// TIA Portal project "Vaja1" (V13)

(* hardware
DEVICE "S7300/ET200M station_1"  S7-300 station
   slot 0: "Rail_0"  Rail  6ES7 390-1***0-0AA0
   slot 1: "PS 307 2A_1"  PS 307 2A  6ES7 307-1BA00-0AA0
   slot 2: "PLC-236"  CPU 315-2 PN/DP  6ES7 315-2EH13-0AB0  V2.6
      slot 1: "MPI/DP interface_1"  X1
      slot 2: "PROFINET interface_1"  PN-IO
         slot 1: "Port_1"  Port
   slot 4: "DI 16/DO 16x24VDC/0.5A_1"  DI16/DO16 x 24V / 0.5A  6ES7 323-1BL00-0AA0
DEVICE "PC station"  SIMATIC PC station
   slot 0: "PC station"  Rail  SIMATIC PC-Station  V1.0
      slot 125: "Stationmanager"  Station_Manager  V6.0.4
   slot 1: "IE general_1"  IE General  IE_CP  V8.2.0
   slot 3: "HMI_RT_1"  WinCC RT Advanced  6AV2 104-0xxxx-xxxx  13.0.1.0
      slot 33792: "Host interface"  Host interface
*)

// ===== PLC "PLC-236"  CPU 315-2 PN/DP =====

VAR_GLOBAL   // PLC tag table "Default tag table"
   "rdeca_levo_potiskac_B_smer_0_nazaj_1_naprej" AT %Q1.4 : Bool;
   "rumena_levo_potiskac_B_premikanje" AT %Q1.5 : Bool;
   "rdeca_desno_tekoci_trak_B_izhod_smer_0_nazaj_1_naprej" AT %Q1.6 : Bool;
   "rumena_desno_tekoci_trak_B_izhod_premikanje" AT %Q1.7 : Bool;
   "kljuc" AT %I1.2 : Bool;
   "zelena" AT %I1.3 : Bool;
   "crna_levo_zgoraj" AT %I1.4 : Bool;
   "crna_levo_spodaj" AT %I1.5 : Bool;
   "crna_desno_zgoraj" AT %I1.6 : Bool;
   "crna_desno_spodaj" AT %I1.7 : Bool;
   "fotocelica_material_na_vhodu_NC" AT %I0.0 : Bool;
   "fotocelica_materal_pred_potiskacem_NC" AT %I0.1 : Bool;
   "potiskac_A_koncni_polozaj_spredaj_NO" AT %I0.2 : Bool;
   "potiskac_A_koncni_polozaj_zadaj_NO" AT %I0.3 : Bool;
   "fotocelica_material_pod_napravo_A_NC" AT %I0.4 : Bool;
   "fotocelica_material_pod_napravo_B_NC" AT %I0.5 : Bool;
   "potiskac_B_koncni_polozaj_zadaj_NO" AT %I0.6 : Bool;
   "potiskac_B_koncni_polozaj_spredaj_NO" AT %I0.7 : Bool;
   "fotocelica_material_na_izhodu_NC" AT %I1.0 : Bool;
   "potiskac_A_smer_0_nazaj_1_naprej" AT %Q0.0 : Bool;
   "potiskac_A_premikanje" AT %Q0.1 : Bool;
   "trak_A_vhod_smer_0_naprej_1_nazaj" AT %Q0.2 : Bool;
   "trak_A_vhod_premikanje" AT %Q0.3 : Bool;
   "trak_A_stroj_smer_0_nazaj_1_naprej" AT %Q0.4 : Bool;
   "trak_A_stroj_premikanje" AT %Q0.5 : Bool;
   "naprava_A_smer_0_CW_1_CCW" AT %Q0.6 : Bool;
   "naprava_A_premikanje" AT %Q0.7 : Bool;
   "naprava_B_smer_0_CW_1_CCW" AT %Q1.0 : Bool;
   "naprava_B_premikanje" AT %Q1.1 : Bool;
   "trak_B_stroj_smer_0_naprej_1_nazaj" AT %Q1.2 : Bool;
   "trak_B_stroj_premikanje" AT %Q1.3 : Bool;
   "retval" AT %MW2 : Int;
   "Startup_Flag" AT %M0.1 : Bool;
   "Ready_Flag" AT %M0.2 : Bool;
   "Clock_10Hz" AT %M5.0 : Bool;
   "Pause_Motors_Flag" AT %M0.3 : Bool;
END_VAR

TYPE "Lokacija"
   STRUCT
      ID : Int;
      zasedenost : Bool;
      senzor : Bool;
      recept : "Recept";
      premikanje : Bool;
   END_STRUCT;
END_TYPE

TYPE "Recept"
   STRUCT
      vrtanje1 : Bool;
      ID_recepta : Int;
      cas_vrtanja1 : Time;
      vrtanje2 : Bool;
      cas_vrtanja2 : Time;
      smer_1 : Bool;
      smer_2 : Bool;
   END_STRUCT;
END_TYPE

// folder: AktivacijaIzvrsnihClenov

DATA_BLOCK "Izhodi"   // DB5
{ S7_Optimized_Access := 'FALSE' }
VERSION : 0.1
   VAR
      potiskac_A_smer : Bool;
      potiskac_A_premikanje : Bool;
      trak_A_vhod_smer : Bool;
      trak_A_vhod_premikanje : Bool;
      trak_A_stroj_smer : Bool;
      trak_A_stroj_premikanje : Bool;
      naprava_A_smer : Bool;
      naprava_A_premikanje : Bool;
      naprava_B_smer : Bool;
      naprava_B_premikanje : Bool;
      trak_B_stroj_smer : Bool;
      trak_B_stroj_premikanje : Bool;
      rdeca_levo_potiskac_B_smer : Bool;
      rumena_levo_potiskac_B_premikanje : Bool;
      rdeca_desno_tekoci_trak_B_izhod_smer : Bool;
      rumena_desno_tekoci_trak_B_izhod_premikanje : Bool;
   END_VAR
BEGIN
END_DATA_BLOCK

// folder: BranjeSenzorjev

DATA_BLOCK "Senzorji_DB"   // DB4
{ S7_Optimized_Access := 'FALSE' }
VERSION : 0.1
   VAR
      fotocelica_material_na_vhodu : Bool;
      fotocelica_materal_pred_potiskacem : Bool;
      navidezni_potiskac_A : Bool;
      potiskac_A_koncni_polozaj_spredaj : Bool;
      potiskac_A_koncni_polozaj_zadaj : Bool;
      fotocelica_material_pod_napravo_A : Bool;
      fotocelica_material_pod_napravo_B : Bool;
      navidezni_potiskac_B : Bool;
      potiskac_B_koncni_polozaj_zadaj : Bool;
      potiskac_B_koncni_polozaj_spredaj : Bool;
      fotocelica_material_na_izhodu : Bool;
      kljuc : Bool;
      zelena_tipka : Bool;
      crna_levo_zgoraj : Bool;
      crna_levo_spodaj : Bool;
      crna_desno_zgoraj : Bool;
      crna_desno_spodaj : Bool;
   END_VAR
BEGIN
END_DATA_BLOCK

// folder: GlavniProgram

DATA_BLOCK "AutoMotorji"   // DB6
{ S7_Optimized_Access := 'FALSE' }
VERSION : 0.1
   VAR
      potiskac_A_naprej : Bool;
      potiskac_A_nazaj : Bool;
      trak_A_vhod_naprej : Bool;
      trak_A_vhod_nazaj : Bool;
      trak_A_stroj_naprej : Bool;
      trak_A_stroj_nazaj : Bool;
      naprava_A_CW : Bool;
      naprava_A_CCW : Bool;
      naprava_B_CW : Bool;
      naprava_B_CCW : Bool;
      trak_B_stroj_naprej : Bool;
      trak_B_stroj_nazaj : Bool;
      potiskac_B_naprej : Bool;
      potiskac_B_nazaj : Bool;
      trak_B_izhod_naprej : Bool;
      trak_B_izhod_nazaj : Bool;
   END_VAR
BEGIN
END_DATA_BLOCK

DATA_BLOCK "Auto_0_vhod1_DB"   // DB8
{ S7_Optimized_Access := 'FALSE' }
VERSION : 0.1
// stored: InstanceOfName Auto_0_vhod1
"Auto_0_vhod1"
BEGIN
END_DATA_BLOCK

DATA_BLOCK "Auto_1_Potiskac_DB"   // DB10
{ S7_Optimized_Access := 'FALSE' }
VERSION : 0.1
// stored: InstanceOfName Auto_1_Potiskac
"Auto_1_Potiskac"
BEGIN
END_DATA_BLOCK

DATA_BLOCK "Auto_2_A_Naprava_DB"   // DB11
{ S7_Optimized_Access := 'FALSE' }
VERSION : 0.1
// stored: InstanceOfName Auto_2_A_Naprava
"Auto_2_A_Naprava"
BEGIN
END_DATA_BLOCK

DATA_BLOCK "Auto_3_B_Naprava_DB"   // DB13
{ S7_Optimized_Access := 'FALSE' }
VERSION : 0.1
// stored: InstanceOfName Auto_3_B_Naprava
"Auto_3_B_Naprava"
BEGIN
END_DATA_BLOCK

DATA_BLOCK "Auto_4_Potiskac_DB"   // DB14
{ S7_Optimized_Access := 'FALSE' }
VERSION : 0.1
// stored: InstanceOfName Auto_4_Potiskac
"Auto_4_Potiskac"
BEGIN
END_DATA_BLOCK

DATA_BLOCK "Auto_5_Izhod_DB"   // DB15
{ S7_Optimized_Access := 'FALSE' }
VERSION : 0.1
// stored: InstanceOfName Auto_5_Izhod
"Auto_5_Izhod"
BEGIN
END_DATA_BLOCK

// folder: GlavniProgram/Alarmi

DATA_BLOCK "Alarmi_DB"   // DB18
{ S7_Optimized_Access := 'FALSE' }
VERSION : 0.1
// stored: InstanceOfName Alarmi
"Alarmi"
BEGIN
END_DATA_BLOCK

// folder: GlavniProgram/SCADA

DATA_BLOCK "SCADA"   // DB16
{ S7_Optimized_Access := 'FALSE' }
VERSION : 0.1
   VAR
      alarmi : Array[0..15] of Bool;
      alarm_aktiven_globalno : Bool;
      recept_num : Int;
      alarm_potrditev : Bool;
      recept : "Recept";
   END_VAR
BEGIN
END_DATA_BLOCK

DATA_BLOCK "SCADAVisual_DB"   // DB23
{ S7_Optimized_Access := 'FALSE' }
VERSION : 0.1
// stored: InstanceOfName SCADAVisual
"SCADAVisual"
BEGIN
END_DATA_BLOCK

// folder: MotorLogic

DATA_BLOCK "Izbira_motorja_DB"   // DB1
{ S7_Optimized_Access := 'FALSE' }
VERSION : 0.1
// stored: InstanceOfName Izbira_motorja
"Izbira_motorja"
BEGIN
END_DATA_BLOCK

DATA_BLOCK "Motorji_DB"   // DB2
{ S7_Optimized_Access := 'FALSE' }
VERSION : 0.1
// stored: InstanceOfName Motorji
"Motorji"
BEGIN
END_DATA_BLOCK

// folder: SledenjeMateriala

DATA_BLOCK "Lokacije_DB"   // DB3
{ S7_Optimized_Access := 'FALSE' }
VERSION : 0.1
   VAR
      L1_vhod_1 : "Lokacija";
      L2_vhod_2 : "Lokacija";
      L3_potiskac_A : "Lokacija";
      L4_naprava_A : "Lokacija";
      L5_naprava_B : "Lokacija";
      L6_potiskac_B : "Lokacija";
      L7_izhod : "Lokacija";
      Empty : "Lokacija";
   END_VAR
BEGIN
END_DATA_BLOCK

// folder: (top level)

ORGANIZATION_BLOCK "Main"   // OB1, LAD
TITLE = "Main Program Sweep (Cycle)"
{ S7_Optimized_Access := 'FALSE' }
VERSION : 0.1
BEGIN

REGION Network 1: Rocno vodenje
   // nc ne bo komentar
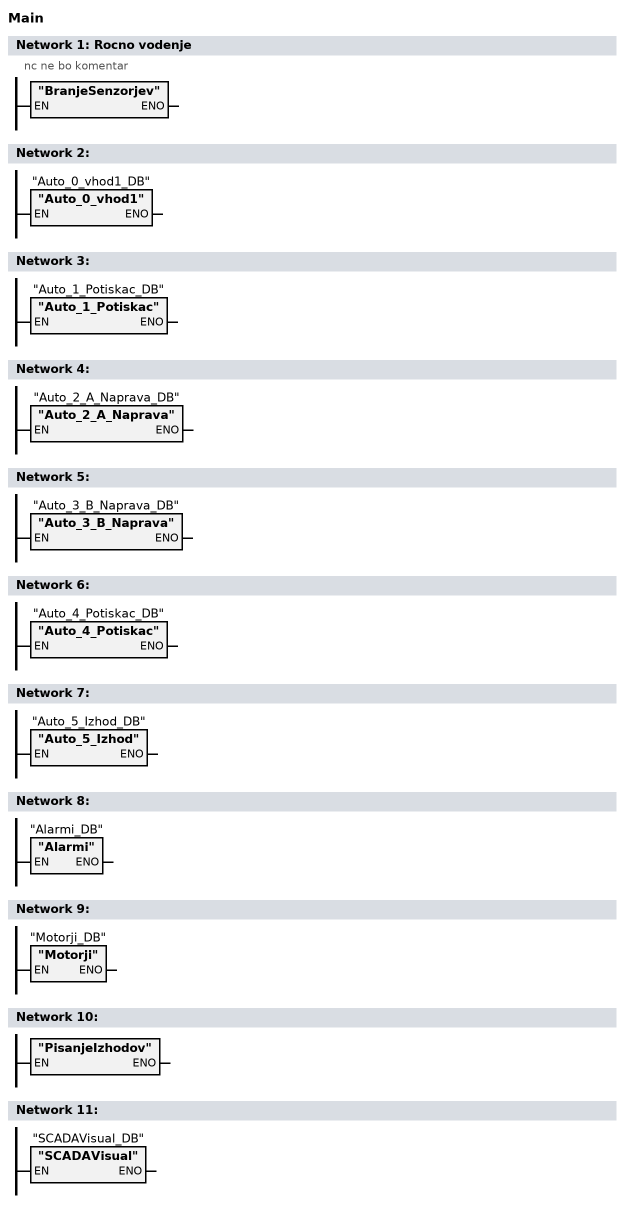
   RUNG wire#powerrail
      "BranjeSenzorjev"()
   END_RUNG
   // the same network as SCL:
   "BranjeSenzorjev"();
END_REGION

REGION Network 2
   RUNG wire#powerrail
      "Auto_0_vhod1_DB"()
   END_RUNG
   // the same network as SCL:
   "Auto_0_vhod1_DB"();   // "Auto_0_vhod1"
END_REGION

REGION Network 3
   RUNG wire#powerrail
      "Auto_1_Potiskac_DB"()
   END_RUNG
   // the same network as SCL:
   "Auto_1_Potiskac_DB"();   // "Auto_1_Potiskac"
END_REGION

REGION Network 4
   RUNG wire#powerrail
      "Auto_2_A_Naprava_DB"()
   END_RUNG
   // the same network as SCL:
   "Auto_2_A_Naprava_DB"();   // "Auto_2_A_Naprava"
END_REGION

REGION Network 5
   RUNG wire#powerrail
      "Auto_3_B_Naprava_DB"()
   END_RUNG
   // the same network as SCL:
   "Auto_3_B_Naprava_DB"();   // "Auto_3_B_Naprava"
END_REGION

REGION Network 6
   RUNG wire#powerrail
      "Auto_4_Potiskac_DB"()
   END_RUNG
   // the same network as SCL:
   "Auto_4_Potiskac_DB"();   // "Auto_4_Potiskac"
END_REGION

REGION Network 7
   RUNG wire#powerrail
      "Auto_5_Izhod_DB"()
   END_RUNG
   // the same network as SCL:
   "Auto_5_Izhod_DB"();   // "Auto_5_Izhod"
END_REGION

REGION Network 8
   RUNG wire#powerrail
      "Alarmi_DB"()
   END_RUNG
   // the same network as SCL:
   "Alarmi_DB"();   // "Alarmi"
END_REGION

REGION Network 9
   RUNG wire#powerrail
      "Motorji_DB"()
   END_RUNG
   // the same network as SCL:
   "Motorji_DB"();   // "Motorji"
END_REGION

REGION Network 10
   RUNG wire#powerrail
      "PisanjeIzhodov"()
   END_RUNG
   // the same network as SCL:
   "PisanjeIzhodov"();
END_REGION

REGION Network 11
   RUNG wire#powerrail
      "SCADAVisual_DB"()
   END_RUNG
   // the same network as SCL:
   "SCADAVisual_DB"();   // "SCADAVisual"
END_REGION
END_ORGANIZATION_BLOCK

// folder: AktivacijaIzvrsnihClenov

FUNCTION "PisanjeIzhodov" : Void   // FC2, LAD
TITLE = Pisanje iz podatkovne baze na izhode.
{ S7_Optimized_Access := 'FALSE' }
VERSION : 0.1
BEGIN

REGION Network 1: Potiskač A smer.
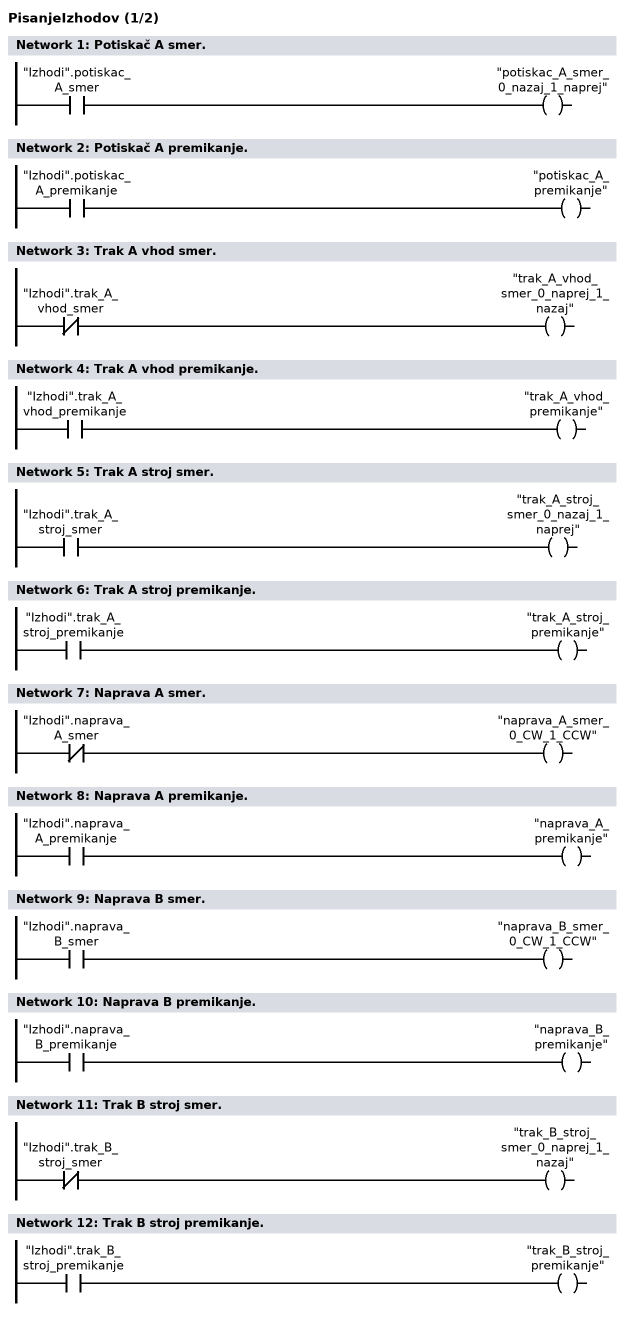
   RUNG wire#powerrail
      Contact( "Izhodi".potiskac_A_smer )
      Coil( "potiskac_A_smer_0_nazaj_1_naprej" )
   END_RUNG
   // the same network as SCL:
   "potiskac_A_smer_0_nazaj_1_naprej" := "Izhodi".potiskac_A_smer;
END_REGION

REGION Network 2: Potiskač A premikanje.
   RUNG wire#powerrail
      Contact( "Izhodi".potiskac_A_premikanje )
      Coil( "potiskac_A_premikanje" )
   END_RUNG
   // the same network as SCL:
   "potiskac_A_premikanje" := "Izhodi".potiskac_A_premikanje;
END_REGION

REGION Network 3: Trak A vhod smer.
   RUNG wire#powerrail
      I_Contact( "Izhodi".trak_A_vhod_smer )
      Coil( "trak_A_vhod_smer_0_naprej_1_nazaj" )
   END_RUNG
   // the same network as SCL:
   "trak_A_vhod_smer_0_naprej_1_nazaj" := NOT "Izhodi".trak_A_vhod_smer;
END_REGION

REGION Network 4: Trak A vhod premikanje.
   RUNG wire#powerrail
      Contact( "Izhodi".trak_A_vhod_premikanje )
      Coil( "trak_A_vhod_premikanje" )
   END_RUNG
   // the same network as SCL:
   "trak_A_vhod_premikanje" := "Izhodi".trak_A_vhod_premikanje;
END_REGION

REGION Network 5: Trak A stroj smer.
   RUNG wire#powerrail
      Contact( "Izhodi".trak_A_stroj_smer )
      Coil( "trak_A_stroj_smer_0_nazaj_1_naprej" )
   END_RUNG
   // the same network as SCL:
   "trak_A_stroj_smer_0_nazaj_1_naprej" := "Izhodi".trak_A_stroj_smer;
END_REGION

REGION Network 6: Trak A stroj premikanje.
   RUNG wire#powerrail
      Contact( "Izhodi".trak_A_stroj_premikanje )
      Coil( "trak_A_stroj_premikanje" )
   END_RUNG
   // the same network as SCL:
   "trak_A_stroj_premikanje" := "Izhodi".trak_A_stroj_premikanje;
END_REGION

REGION Network 7: Naprava A smer.
   RUNG wire#powerrail
      I_Contact( "Izhodi".naprava_A_smer )
      Coil( "naprava_A_smer_0_CW_1_CCW" )
   END_RUNG
   // the same network as SCL:
   "naprava_A_smer_0_CW_1_CCW" := NOT "Izhodi".naprava_A_smer;
END_REGION

REGION Network 8: Naprava A premikanje.
   RUNG wire#powerrail
      Contact( "Izhodi".naprava_A_premikanje )
      Coil( "naprava_A_premikanje" )
   END_RUNG
   // the same network as SCL:
   "naprava_A_premikanje" := "Izhodi".naprava_A_premikanje;
END_REGION

REGION Network 9: Naprava B smer.
   RUNG wire#powerrail
      Contact( "Izhodi".naprava_B_smer )
      Coil( "naprava_B_smer_0_CW_1_CCW" )
   END_RUNG
   // the same network as SCL:
   "naprava_B_smer_0_CW_1_CCW" := "Izhodi".naprava_B_smer;
END_REGION

REGION Network 10: Naprava B premikanje.
   RUNG wire#powerrail
      Contact( "Izhodi".naprava_B_premikanje )
      Coil( "naprava_B_premikanje" )
   END_RUNG
   // the same network as SCL:
   "naprava_B_premikanje" := "Izhodi".naprava_B_premikanje;
END_REGION

REGION Network 11: Trak B stroj smer.
   RUNG wire#powerrail
      I_Contact( "Izhodi".trak_B_stroj_smer )
      Coil( "trak_B_stroj_smer_0_naprej_1_nazaj" )
   END_RUNG
   // the same network as SCL:
   "trak_B_stroj_smer_0_naprej_1_nazaj" := NOT "Izhodi".trak_B_stroj_smer;
END_REGION

REGION Network 12: Trak B stroj premikanje.
   RUNG wire#powerrail
      Contact( "Izhodi".trak_B_stroj_premikanje )
      Coil( "trak_B_stroj_premikanje" )
   END_RUNG
   // the same network as SCL:
   "trak_B_stroj_premikanje" := "Izhodi".trak_B_stroj_premikanje;
END_REGION

REGION Network 13: Potiskač B smer.
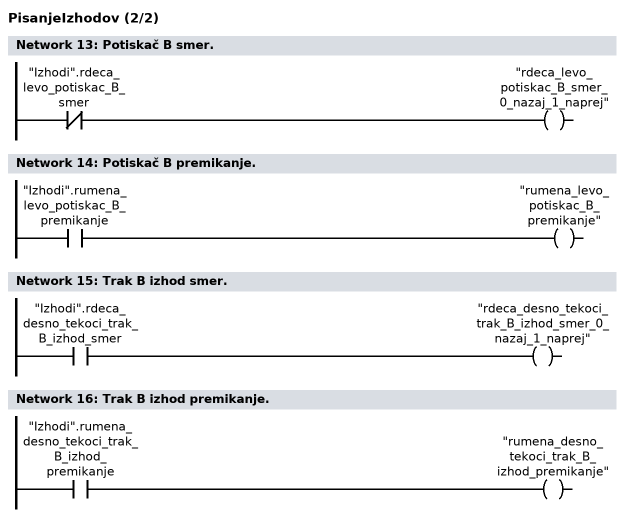
   RUNG wire#powerrail
      I_Contact( "Izhodi".rdeca_levo_potiskac_B_smer )
      Coil( "rdeca_levo_potiskac_B_smer_0_nazaj_1_naprej" )
   END_RUNG
   // the same network as SCL:
   "rdeca_levo_potiskac_B_smer_0_nazaj_1_naprej" := NOT "Izhodi".rdeca_levo_potiskac_B_smer;
END_REGION

REGION Network 14: Potiskač B premikanje.
   RUNG wire#powerrail
      Contact( "Izhodi".rumena_levo_potiskac_B_premikanje )
      Coil( "rumena_levo_potiskac_B_premikanje" )
   END_RUNG
   // the same network as SCL:
   "rumena_levo_potiskac_B_premikanje" := "Izhodi".rumena_levo_potiskac_B_premikanje;
END_REGION

REGION Network 15: Trak B izhod smer.
   RUNG wire#powerrail
      Contact( "Izhodi".rdeca_desno_tekoci_trak_B_izhod_smer )
      Coil( "rdeca_desno_tekoci_trak_B_izhod_smer_0_nazaj_1_naprej" )
   END_RUNG
   // the same network as SCL:
   "rdeca_desno_tekoci_trak_B_izhod_smer_0_nazaj_1_naprej" := "Izhodi".rdeca_desno_tekoci_trak_B_izhod_smer;
END_REGION

REGION Network 16: Trak B izhod premikanje.
   RUNG wire#powerrail
      Contact( "Izhodi".rumena_desno_tekoci_trak_B_izhod_premikanje )
      Coil( "rumena_desno_tekoci_trak_B_izhod_premikanje" )
   END_RUNG
   // the same network as SCL:
   "rumena_desno_tekoci_trak_B_izhod_premikanje" := "Izhodi".rumena_desno_tekoci_trak_B_izhod_premikanje;
END_REGION
END_FUNCTION

// folder: BranjeSenzorjev

FUNCTION "BranjeSenzorjev" : Void   // FC1, LAD
TITLE = Prepis iz vhodov v podatkovno bazo.
{ S7_Optimized_Access := 'FALSE' }
VERSION : 0.1
// Normaliziranje vseh senzorjev (NC/NO).
BEGIN

REGION Network 1: Fotocelica: material na vhodu.
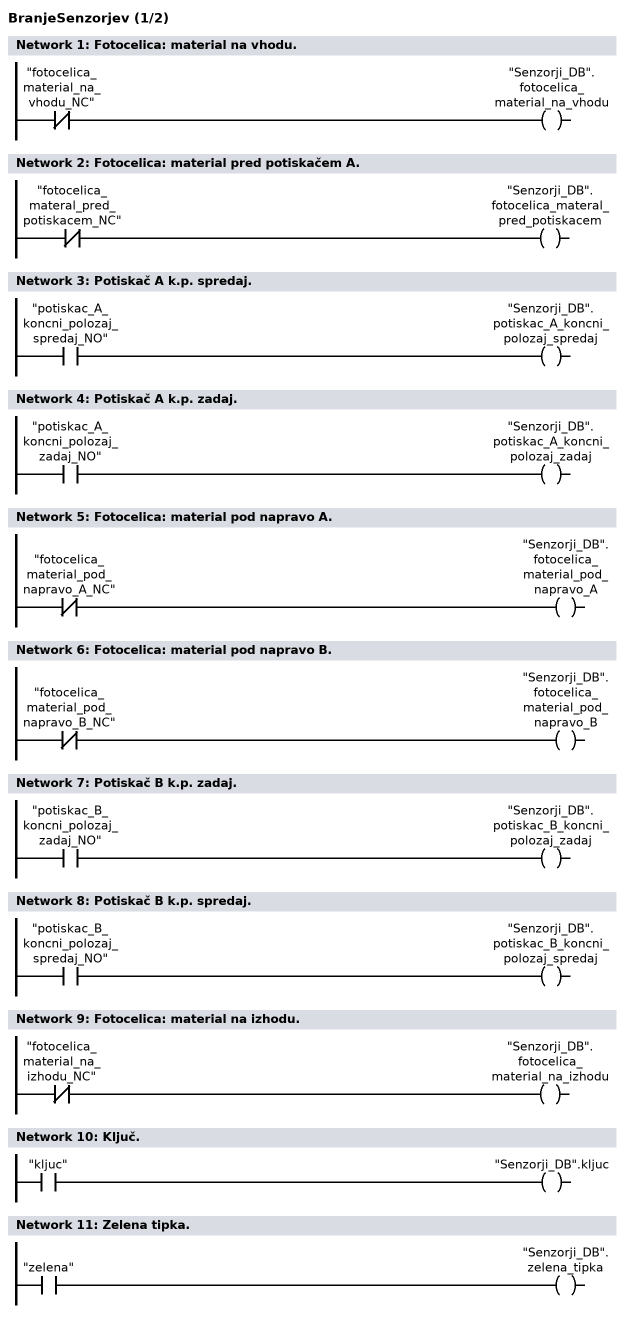
   RUNG wire#powerrail
      I_Contact( "fotocelica_material_na_vhodu_NC" )
      Coil( "Senzorji_DB".fotocelica_material_na_vhodu )
   END_RUNG
   // the same network as SCL:
   "Senzorji_DB".fotocelica_material_na_vhodu := NOT "fotocelica_material_na_vhodu_NC";
END_REGION

REGION Network 2: Fotocelica: material pred potiskačem A.
   RUNG wire#powerrail
      I_Contact( "fotocelica_materal_pred_potiskacem_NC" )
      Coil( "Senzorji_DB".fotocelica_materal_pred_potiskacem )
   END_RUNG
   // the same network as SCL:
   "Senzorji_DB".fotocelica_materal_pred_potiskacem := NOT "fotocelica_materal_pred_potiskacem_NC";
END_REGION

REGION Network 3: Potiskač A k.p. spredaj.
   RUNG wire#powerrail
      Contact( "potiskac_A_koncni_polozaj_spredaj_NO" )
      Coil( "Senzorji_DB".potiskac_A_koncni_polozaj_spredaj )
   END_RUNG
   // the same network as SCL:
   "Senzorji_DB".potiskac_A_koncni_polozaj_spredaj := "potiskac_A_koncni_polozaj_spredaj_NO";
END_REGION

REGION Network 4: Potiskač A k.p. zadaj.
   RUNG wire#powerrail
      Contact( "potiskac_A_koncni_polozaj_zadaj_NO" )
      Coil( "Senzorji_DB".potiskac_A_koncni_polozaj_zadaj )
   END_RUNG
   // the same network as SCL:
   "Senzorji_DB".potiskac_A_koncni_polozaj_zadaj := "potiskac_A_koncni_polozaj_zadaj_NO";
END_REGION

REGION Network 5: Fotocelica: material pod napravo A.
   RUNG wire#powerrail
      I_Contact( "fotocelica_material_pod_napravo_A_NC" )
      Coil( "Senzorji_DB".fotocelica_material_pod_napravo_A )
   END_RUNG
   // the same network as SCL:
   "Senzorji_DB".fotocelica_material_pod_napravo_A := NOT "fotocelica_material_pod_napravo_A_NC";
END_REGION

REGION Network 6: Fotocelica: material pod napravo B.
   RUNG wire#powerrail
      I_Contact( "fotocelica_material_pod_napravo_B_NC" )
      Coil( "Senzorji_DB".fotocelica_material_pod_napravo_B )
   END_RUNG
   // the same network as SCL:
   "Senzorji_DB".fotocelica_material_pod_napravo_B := NOT "fotocelica_material_pod_napravo_B_NC";
END_REGION

REGION Network 7: Potiskač B k.p. zadaj.
   RUNG wire#powerrail
      Contact( "potiskac_B_koncni_polozaj_zadaj_NO" )
      Coil( "Senzorji_DB".potiskac_B_koncni_polozaj_zadaj )
   END_RUNG
   // the same network as SCL:
   "Senzorji_DB".potiskac_B_koncni_polozaj_zadaj := "potiskac_B_koncni_polozaj_zadaj_NO";
END_REGION

REGION Network 8: Potiskač B k.p. spredaj.
   RUNG wire#powerrail
      Contact( "potiskac_B_koncni_polozaj_spredaj_NO" )
      Coil( "Senzorji_DB".potiskac_B_koncni_polozaj_spredaj )
   END_RUNG
   // the same network as SCL:
   "Senzorji_DB".potiskac_B_koncni_polozaj_spredaj := "potiskac_B_koncni_polozaj_spredaj_NO";
END_REGION

REGION Network 9: Fotocelica: material na izhodu.
   RUNG wire#powerrail
      I_Contact( "fotocelica_material_na_izhodu_NC" )
      Coil( "Senzorji_DB".fotocelica_material_na_izhodu )
   END_RUNG
   // the same network as SCL:
   "Senzorji_DB".fotocelica_material_na_izhodu := NOT "fotocelica_material_na_izhodu_NC";
END_REGION

REGION Network 10: Ključ.
   RUNG wire#powerrail
      Contact( "kljuc" )
      Coil( "Senzorji_DB".kljuc )
   END_RUNG
   // the same network as SCL:
   "Senzorji_DB".kljuc := "kljuc";
END_REGION

REGION Network 11: Zelena tipka.
   RUNG wire#powerrail
      Contact( "zelena" )
      Coil( "Senzorji_DB".zelena_tipka )
   END_RUNG
   // the same network as SCL:
   "Senzorji_DB".zelena_tipka := "zelena";
END_REGION

REGION Network 12: Črna tipka levo zgoraj.
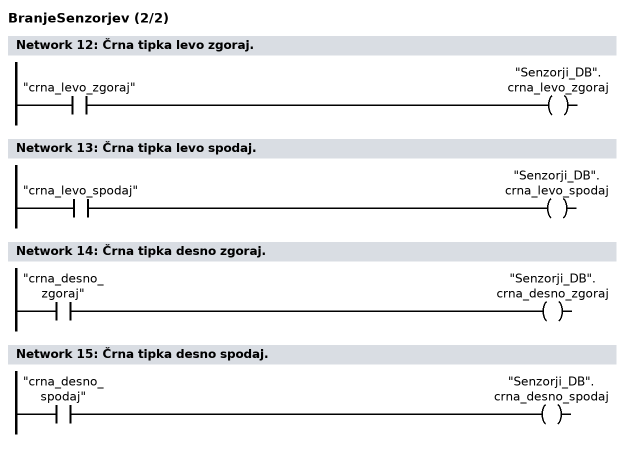
   RUNG wire#powerrail
      Contact( "crna_levo_zgoraj" )
      Coil( "Senzorji_DB".crna_levo_zgoraj )
   END_RUNG
   // the same network as SCL:
   "Senzorji_DB".crna_levo_zgoraj := "crna_levo_zgoraj";
END_REGION

REGION Network 13: Črna tipka levo spodaj.
   RUNG wire#powerrail
      Contact( "crna_levo_spodaj" )
      Coil( "Senzorji_DB".crna_levo_spodaj )
   END_RUNG
   // the same network as SCL:
   "Senzorji_DB".crna_levo_spodaj := "crna_levo_spodaj";
END_REGION

REGION Network 14: Črna tipka desno zgoraj.
   RUNG wire#powerrail
      Contact( "crna_desno_zgoraj" )
      Coil( "Senzorji_DB".crna_desno_zgoraj )
   END_RUNG
   // the same network as SCL:
   "Senzorji_DB".crna_desno_zgoraj := "crna_desno_zgoraj";
END_REGION

REGION Network 15: Črna tipka desno spodaj.
   RUNG wire#powerrail
      Contact( "crna_desno_spodaj" )
      Coil( "Senzorji_DB".crna_desno_spodaj )
   END_RUNG
   // the same network as SCL:
   "Senzorji_DB".crna_desno_spodaj := "crna_desno_spodaj";
END_REGION
END_FUNCTION

// folder: GlavniProgram

FUNCTION_BLOCK "Auto_2_A_Naprava"   // FB4, LAD
TITLE = Stanje 2: Naprava A.
{ S7_Optimized_Access := 'FALSE' }
VERSION : 0.1
// V stanju dve vrtimo napravo A za čas definiran v receptu in smer definirano v receptu, potem material pošljemo do naprave B.
   VAR_TEMP   // added for the SCL form of the ladder/FBD networks
      _w1 : Bool;
      _w2 : Bool;
      _w3 : Bool;
      _w4 : Bool;
      _w5 : Bool;
   END_VAR
BEGIN

REGION Network 1
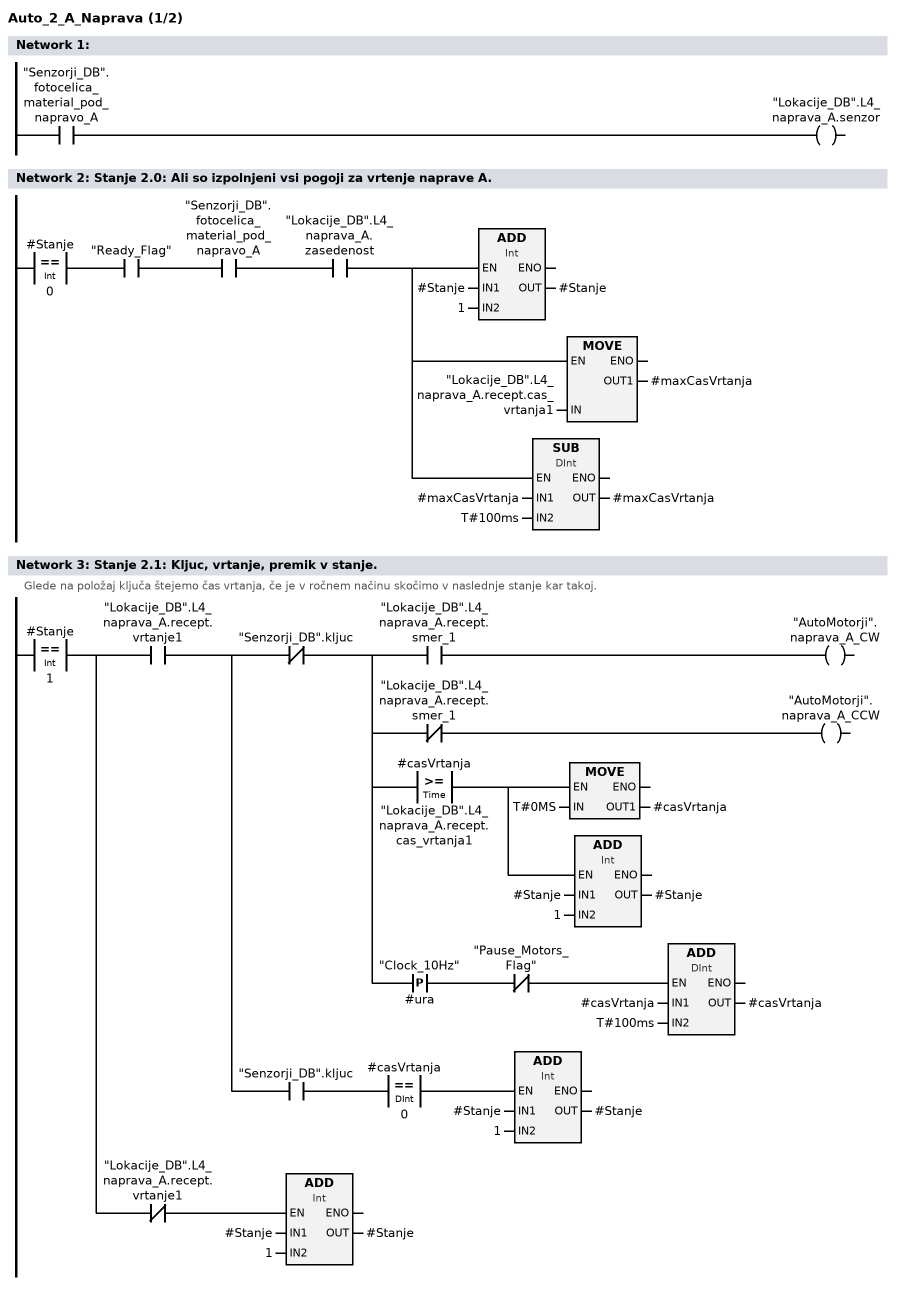
   RUNG wire#powerrail
      Contact( "Senzorji_DB".fotocelica_material_pod_napravo_A )
      Coil( "Lokacije_DB".L4_naprava_A.senzor )
   END_RUNG
   // the same network as SCL:
   "Lokacije_DB".L4_naprava_A.senzor := "Senzorji_DB".fotocelica_material_pod_napravo_A;
END_REGION

REGION Network 2: Stanje 2.0: Ali so izpolnjeni vsi pogoji za vrtenje naprave A.
   RUNG wire#powerrail
      { S7_Templates := "SrcType := Int" } EQ_Contact(in1 := #Stanje, in2 := 0)
      Contact( "Ready_Flag" )
      Contact( "Senzorji_DB".fotocelica_material_pod_napravo_A )
      Contact( "Lokacije_DB".L4_naprava_A.zasedenost )
      wire#w1
      { S7_Templates := "SrcType := Int"; S7_GenerateENO := "TRUE" } Add(in1 := #Stanje, in2 := 1, out => #Stanje)
   END_RUNG
   RUNG wire#w1
      { S7_GenerateENO := "TRUE" } Move(in := "Lokacije_DB".L4_naprava_A.recept.cas_vrtanja1, out1 => #maxCasVrtanja)
   END_RUNG
   RUNG wire#w1
      { S7_Templates := "SrcType := DInt"; S7_GenerateENO := "TRUE" } Sub(in1 := #maxCasVrtanja, in2 := T#100ms, out => #maxCasVrtanja)
   END_RUNG
   // the same network as SCL:
   #_w1 := (#Stanje = 0) AND "Ready_Flag" AND "Senzorji_DB".fotocelica_material_pod_napravo_A AND "Lokacije_DB".L4_naprava_A.zasedenost;
   IF #_w1 THEN
       #Stanje := #Stanje + 1;
       #maxCasVrtanja := "Lokacije_DB".L4_naprava_A.recept.cas_vrtanja1;
       #maxCasVrtanja := #maxCasVrtanja - T#100ms;
   END_IF;
END_REGION

REGION Network 3: Stanje 2.1: Kljuc, vrtanje, premik v stanje.
   // Glede na položaj ključa štejemo čas vrtanja, če je v ročnem načinu skočimo v naslednje stanje kar takoj.
   RUNG wire#powerrail
      { S7_Templates := "SrcType := Int" } EQ_Contact(in1 := #Stanje, in2 := 1)
      wire#w1
      Contact( "Lokacije_DB".L4_naprava_A.recept.vrtanje1 )
      wire#w2
      I_Contact( "Senzorji_DB".kljuc )
      wire#w3
      Contact( "Lokacije_DB".L4_naprava_A.recept.smer_1 )
      Coil( "AutoMotorji".naprava_A_CW )
   END_RUNG
   RUNG wire#w3
      I_Contact( "Lokacije_DB".L4_naprava_A.recept.smer_1 )
      Coil( "AutoMotorji".naprava_A_CCW )
   END_RUNG
   RUNG wire#w3
      { S7_Templates := "SrcType := Time" } GE_Contact(in1 := #casVrtanja, in2 := "Lokacije_DB".L4_naprava_A.recept.cas_vrtanja1)
      wire#w4
      { S7_GenerateENO := "TRUE" } Move(in := T#0MS, out1 => #casVrtanja)
   END_RUNG
   RUNG wire#w4
      { S7_Templates := "SrcType := Int"; S7_GenerateENO := "TRUE" } Add(in1 := #Stanje, in2 := 1, out => #Stanje)
   END_RUNG
   RUNG wire#w3
      P_Contact(operand := "Clock_10Hz", bit := #ura)
      I_Contact( "Pause_Motors_Flag" )
      { S7_Templates := "SrcType := DInt"; S7_GenerateENO := "TRUE" } Add(in1 := #casVrtanja, in2 := T#100ms, out => #casVrtanja)
   END_RUNG
   RUNG wire#w2
      Contact( "Senzorji_DB".kljuc )
      { S7_Templates := "SrcType := DInt" } EQ_Contact(in1 := #casVrtanja, in2 := 0)
      { S7_Templates := "SrcType := Int"; S7_GenerateENO := "TRUE" } Add(in1 := #Stanje, in2 := 1, out => #Stanje)
   END_RUNG
   RUNG wire#w1
      I_Contact( "Lokacije_DB".L4_naprava_A.recept.vrtanje1 )
      { S7_Templates := "SrcType := Int"; S7_GenerateENO := "TRUE" } Add(in1 := #Stanje, in2 := 1, out => #Stanje)
   END_RUNG
   // the same network as SCL:
   #_w1 := #Stanje = 1;
   #_w2 := #_w1 AND "Lokacije_DB".L4_naprava_A.recept.vrtanje1;
   #_w3 := #_w2 AND NOT "Senzorji_DB".kljuc;
   "AutoMotorji".naprava_A_CW := #_w3 AND "Lokacije_DB".L4_naprava_A.recept.smer_1;
   "AutoMotorji".naprava_A_CCW := #_w3 AND NOT "Lokacije_DB".L4_naprava_A.recept.smer_1;
   #_w4 := #_w3 AND (#casVrtanja >= "Lokacije_DB".L4_naprava_A.recept.cas_vrtanja1);
   IF #_w4 THEN
       #casVrtanja := T#0MS;
       #Stanje := #Stanje + 1;
   END_IF;
   #_w5 := #_w3 AND "Clock_10Hz" AND NOT #ura;   // rising edge of "Clock_10Hz"
   #ura := "Clock_10Hz";
   IF #_w5 AND NOT "Pause_Motors_Flag" THEN #casVrtanja := #casVrtanja + T#100ms; END_IF;
   IF #_w2 AND "Senzorji_DB".kljuc AND (#casVrtanja = 0) THEN #Stanje := #Stanje + 1; END_IF;
   IF #_w1 AND NOT "Lokacije_DB".L4_naprava_A.recept.vrtanje1 THEN #Stanje := #Stanje + 1; END_IF;
END_REGION

REGION Network 4: Stanje 2.2: Po koncu vrtanja prižgemo tekoča traka, da pride material pod napravo B.
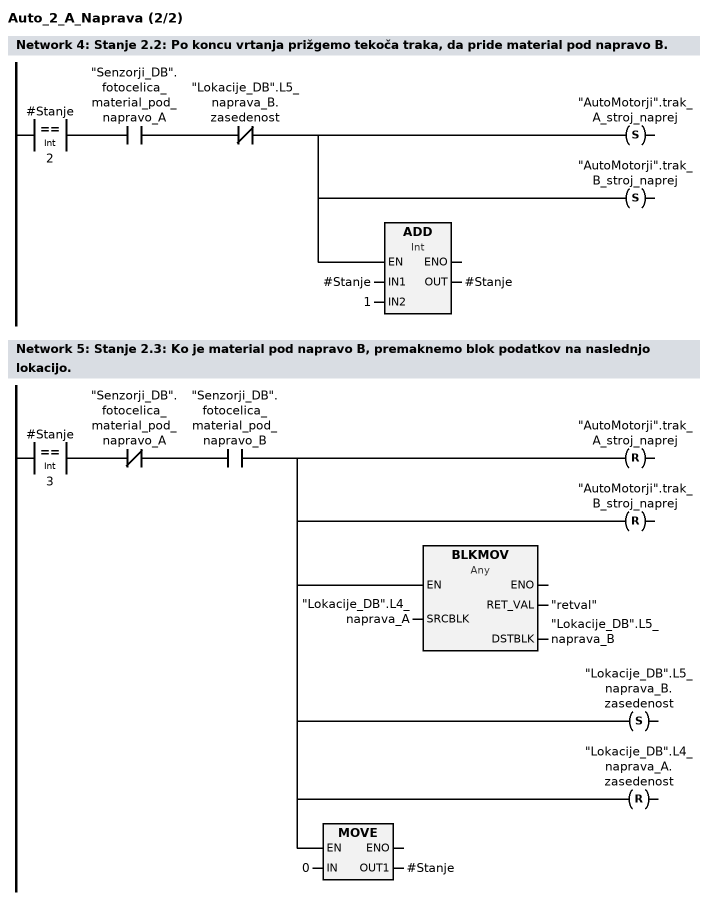
   RUNG wire#powerrail
      { S7_Templates := "SrcType := Int" } EQ_Contact(in1 := #Stanje, in2 := 2)
      Contact( "Senzorji_DB".fotocelica_material_pod_napravo_A )
      I_Contact( "Lokacije_DB".L5_naprava_B.zasedenost )
      wire#w1
      S_Coil( "AutoMotorji".trak_A_stroj_naprej )
   END_RUNG
   RUNG wire#w1
      S_Coil( "AutoMotorji".trak_B_stroj_naprej )
   END_RUNG
   RUNG wire#w1
      { S7_Templates := "SrcType := Int"; S7_GenerateENO := "TRUE" } Add(in1 := #Stanje, in2 := 1, out => #Stanje)
   END_RUNG
   // the same network as SCL:
   IF (#Stanje = 2) AND "Senzorji_DB".fotocelica_material_pod_napravo_A AND NOT "Lokacije_DB".L5_naprava_B.zasedenost THEN
       "AutoMotorji".trak_A_stroj_naprej := TRUE;
       "AutoMotorji".trak_B_stroj_naprej := TRUE;
       #Stanje := #Stanje + 1;
   END_IF;
END_REGION

REGION Network 5: Stanje 2.3: Ko je material pod napravo B, premaknemo blok podatkov na naslednjo lokacijo.
   IF (#Stanje = 3) AND NOT "Senzorji_DB".fotocelica_material_pod_napravo_A AND "Senzorji_DB".fotocelica_material_pod_napravo_B THEN
       "AutoMotorji".trak_A_stroj_naprej := FALSE;
       "AutoMotorji".trak_B_stroj_naprej := FALSE;
   END_IF;
   #_w1 := (#Stanje = 3) AND NOT "Senzorji_DB".fotocelica_material_pod_napravo_A AND "Senzorji_DB".fotocelica_material_pod_napravo_B;
   IF #_w1 THEN
       "retval" := BLKMOV(SRCBLK := "Lokacije_DB".L4_naprava_A, DSTBLK => "Lokacije_DB".L5_naprava_B);
       "Lokacije_DB".L5_naprava_B.zasedenost := TRUE;
       "Lokacije_DB".L4_naprava_A.zasedenost := FALSE;
       #Stanje := 0;
   END_IF;
END_REGION
END_FUNCTION_BLOCK

FUNCTION_BLOCK "Auto_1_Potiskac"   // FB5, LAD
TITLE = Stanje 1 -> potiskač
{ S7_Optimized_Access := 'FALSE' }
VERSION : 0.1
// Premikanje materiala izpred potiskača do drugega tekočega traku.
   VAR_TEMP   // added for the SCL form of the ladder/FBD networks
      _w1 : Bool;
      _w2 : Bool;
      _w3 : Bool;
      _w4 : Bool;
   END_VAR
BEGIN

REGION Network 1: Stanje 1.0: Preverimo ali so vsi pogoji ustrezni za premikanje potiskača.
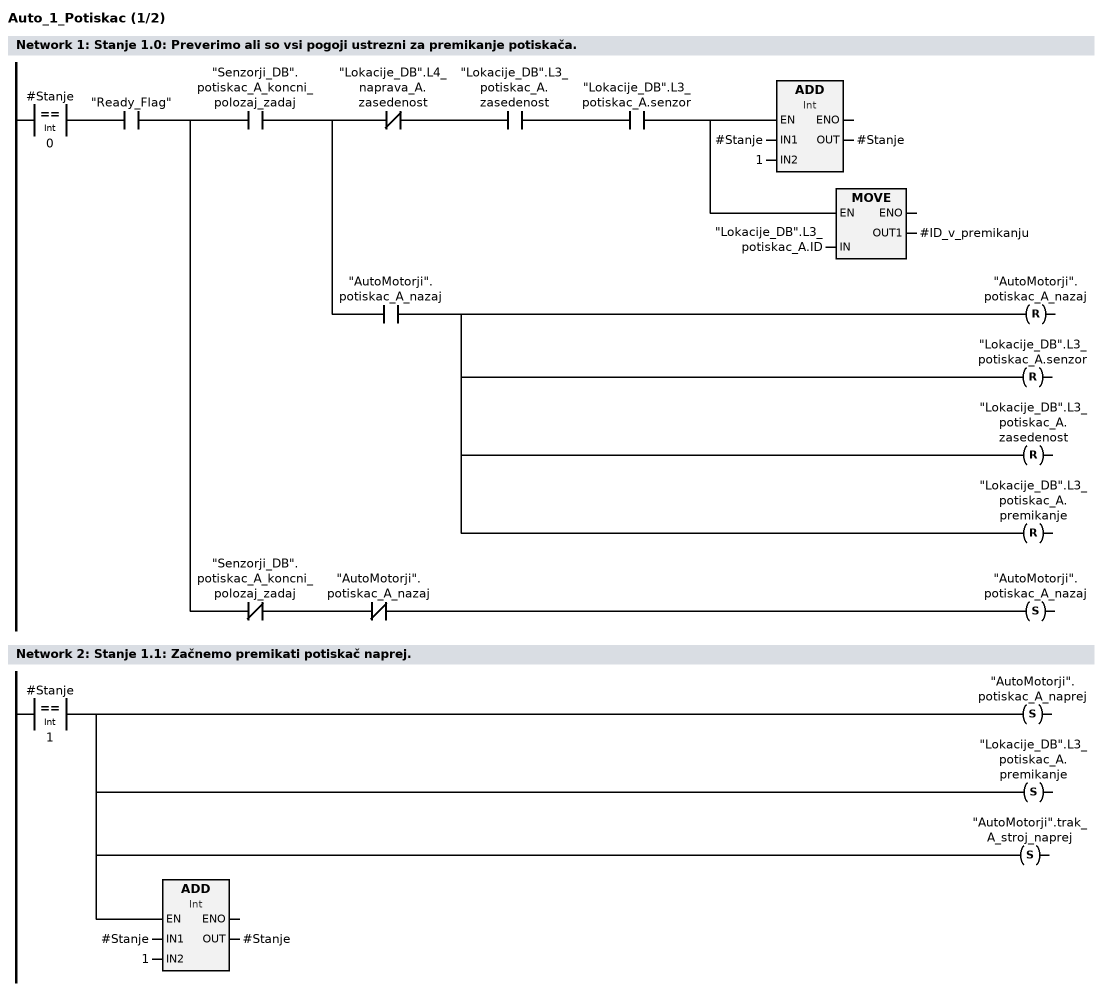
   RUNG wire#powerrail
      { S7_Templates := "SrcType := Int" } EQ_Contact(in1 := #Stanje, in2 := 0)
      Contact( "Ready_Flag" )
      wire#w1
      Contact( "Senzorji_DB".potiskac_A_koncni_polozaj_zadaj )
      wire#w2
      I_Contact( "Lokacije_DB".L4_naprava_A.zasedenost )
      Contact( "Lokacije_DB".L3_potiskac_A.zasedenost )
      Contact( "Lokacije_DB".L3_potiskac_A.senzor )
      wire#w3
      { S7_Templates := "SrcType := Int"; S7_GenerateENO := "TRUE" } Add(in1 := #Stanje, in2 := 1, out => #Stanje)
   END_RUNG
   RUNG wire#w3
      { S7_GenerateENO := "TRUE" } Move(in := "Lokacije_DB".L3_potiskac_A.ID, out1 => #ID_v_premikanju)
   END_RUNG
   RUNG wire#w2
      Contact( "AutoMotorji".potiskac_A_nazaj )
      wire#w4
      R_Coil( "AutoMotorji".potiskac_A_nazaj )
   END_RUNG
   RUNG wire#w4
      R_Coil( "Lokacije_DB".L3_potiskac_A.senzor )
   END_RUNG
   RUNG wire#w4
      R_Coil( "Lokacije_DB".L3_potiskac_A.zasedenost )
   END_RUNG
   RUNG wire#w4
      R_Coil( "Lokacije_DB".L3_potiskac_A.premikanje )
   END_RUNG
   RUNG wire#w1
      I_Contact( "Senzorji_DB".potiskac_A_koncni_polozaj_zadaj )
      I_Contact( "AutoMotorji".potiskac_A_nazaj )
      S_Coil( "AutoMotorji".potiskac_A_nazaj )
   END_RUNG
   // the same network as SCL:
   #_w1 := (#Stanje = 0) AND "Ready_Flag";
   #_w2 := #_w1 AND "Senzorji_DB".potiskac_A_koncni_polozaj_zadaj;
   IF #_w2 AND NOT "Lokacije_DB".L4_naprava_A.zasedenost AND "Lokacije_DB".L3_potiskac_A.zasedenost AND "Lokacije_DB".L3_potiskac_A.senzor THEN
       #Stanje := #Stanje + 1;
       #ID_v_premikanju := "Lokacije_DB".L3_potiskac_A.ID;
   END_IF;
   #_w3 := #_w2 AND "AutoMotorji".potiskac_A_nazaj;
   IF #_w3 THEN
       "AutoMotorji".potiskac_A_nazaj := FALSE;
       "Lokacije_DB".L3_potiskac_A.senzor := FALSE;
       "Lokacije_DB".L3_potiskac_A.zasedenost := FALSE;
       "Lokacije_DB".L3_potiskac_A.premikanje := FALSE;
   END_IF;
   IF #_w1 AND NOT "Senzorji_DB".potiskac_A_koncni_polozaj_zadaj AND NOT "AutoMotorji".potiskac_A_nazaj THEN
       "AutoMotorji".potiskac_A_nazaj := TRUE;
   END_IF;
END_REGION

REGION Network 2: Stanje 1.1: Začnemo premikati potiskač naprej.
   RUNG wire#powerrail
      { S7_Templates := "SrcType := Int" } EQ_Contact(in1 := #Stanje, in2 := 1)
      wire#w1
      S_Coil( "AutoMotorji".potiskac_A_naprej )
   END_RUNG
   RUNG wire#w1
      S_Coil( "Lokacije_DB".L3_potiskac_A.premikanje )
   END_RUNG
   RUNG wire#w1
      S_Coil( "AutoMotorji".trak_A_stroj_naprej )
   END_RUNG
   RUNG wire#w1
      { S7_Templates := "SrcType := Int"; S7_GenerateENO := "TRUE" } Add(in1 := #Stanje, in2 := 1, out => #Stanje)
   END_RUNG
   // the same network as SCL:
   IF #Stanje = 1 THEN
       "AutoMotorji".potiskac_A_naprej := TRUE;
       "Lokacije_DB".L3_potiskac_A.premikanje := TRUE;
       "AutoMotorji".trak_A_stroj_naprej := TRUE;
       #Stanje := #Stanje + 1;
   END_IF;
END_REGION

REGION Network 3: Stanje 1.2: Potiskač A naprej, tekoči trak, fotocelica, potiskač nazaj.
   // Premikamo potiskač A naprej in vrtimo tekoči trak, dokler ne pride material pod fotocelico, potem premaknemo potiskač nazaj,
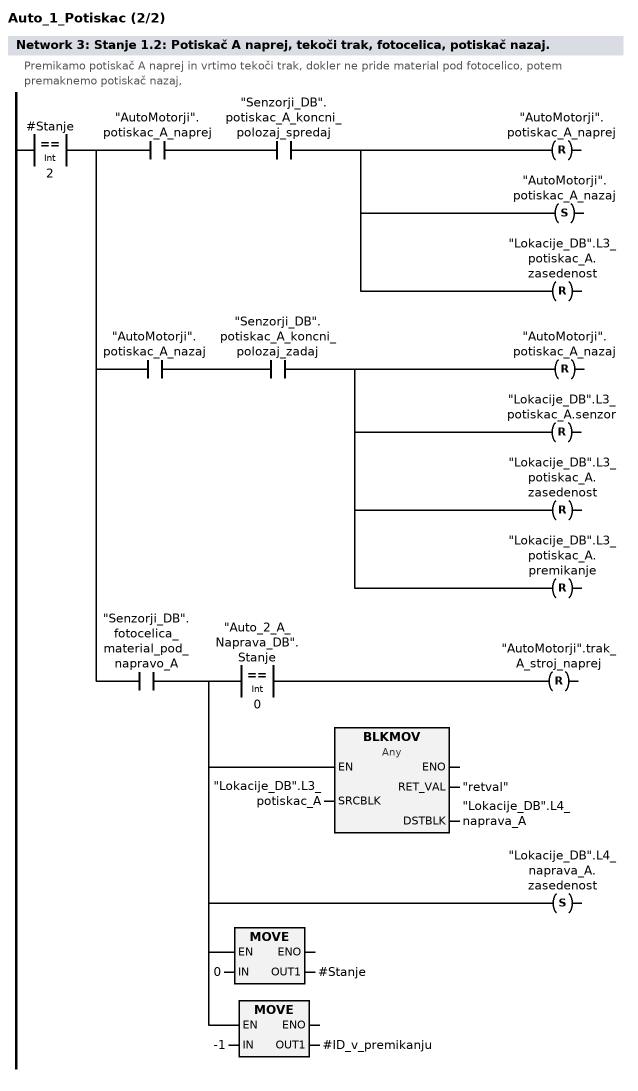
   #_w1 := #Stanje = 2;
   #_w2 := #_w1 AND "AutoMotorji".potiskac_A_naprej AND "Senzorji_DB".potiskac_A_koncni_polozaj_spredaj;
   IF #_w2 THEN
       "AutoMotorji".potiskac_A_naprej := FALSE;
       "AutoMotorji".potiskac_A_nazaj := TRUE;
       "Lokacije_DB".L3_potiskac_A.zasedenost := FALSE;
   END_IF;
   #_w3 := #_w1 AND "AutoMotorji".potiskac_A_nazaj AND "Senzorji_DB".potiskac_A_koncni_polozaj_zadaj;
   IF #_w3 THEN
       "AutoMotorji".potiskac_A_nazaj := FALSE;
       "Lokacije_DB".L3_potiskac_A.senzor := FALSE;
       "Lokacije_DB".L3_potiskac_A.zasedenost := FALSE;
       "Lokacije_DB".L3_potiskac_A.premikanje := FALSE;
   END_IF;
   #_w4 := #_w1 AND "Senzorji_DB".fotocelica_material_pod_napravo_A;
   IF #_w4 AND ("Auto_2_A_Naprava_DB".Stanje = 0) THEN "AutoMotorji".trak_A_stroj_naprej := FALSE; END_IF;
   IF #_w4 THEN
       "retval" := BLKMOV(SRCBLK := "Lokacije_DB".L3_potiskac_A, DSTBLK => "Lokacije_DB".L4_naprava_A);
       "Lokacije_DB".L4_naprava_A.zasedenost := TRUE;
       #Stanje := 0;
       #ID_v_premikanju := -1;
   END_IF;
END_REGION
END_FUNCTION_BLOCK

FUNCTION_BLOCK "Auto_0_vhod1"   // FB6, LAD
TITLE = Stanje 0 -> vhod na tekoči trak; 1. in 2. fotocelica
{ S7_Optimized_Access := 'FALSE' }
VERSION : 0.1
// Program za generiranje recepta, vhod na linijo z dvema napravama, obsega tekoči trak in prvi dve fotocelici.
   VAR_TEMP   // added for the SCL form of the ladder/FBD networks
      _w1 : Bool;
      _w2 : Bool;
   END_VAR
BEGIN

REGION Network 1: Prepis stanja fotocelice v Lokacije DB.
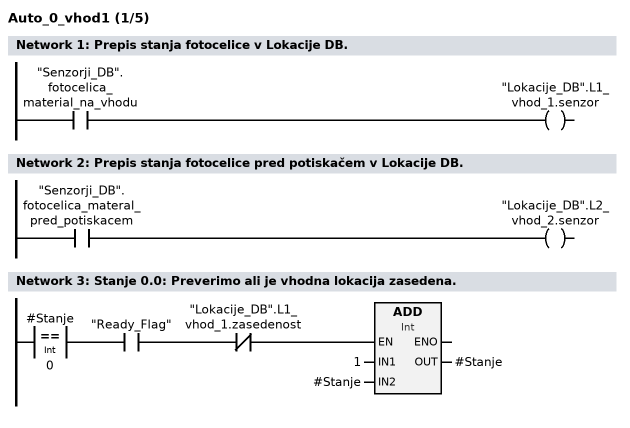
   RUNG wire#powerrail
      Contact( "Senzorji_DB".fotocelica_material_na_vhodu )
      Coil( "Lokacije_DB".L1_vhod_1.senzor )
   END_RUNG
   // the same network as SCL:
   "Lokacije_DB".L1_vhod_1.senzor := "Senzorji_DB".fotocelica_material_na_vhodu;
END_REGION

REGION Network 2: Prepis stanja fotocelice pred potiskačem v Lokacije DB.
   RUNG wire#powerrail
      Contact( "Senzorji_DB".fotocelica_materal_pred_potiskacem )
      Coil( "Lokacije_DB".L2_vhod_2.senzor )
   END_RUNG
   // the same network as SCL:
   "Lokacije_DB".L2_vhod_2.senzor := "Senzorji_DB".fotocelica_materal_pred_potiskacem;
END_REGION

REGION Network 3: Stanje 0.0: Preverimo ali je vhodna lokacija zasedena.
   RUNG wire#powerrail
      { S7_Templates := "SrcType := Int" } EQ_Contact(in1 := #Stanje, in2 := 0)
      Contact( "Ready_Flag" )
      I_Contact( "Lokacije_DB".L1_vhod_1.zasedenost )
      { S7_Templates := "SrcType := Int"; S7_GenerateENO := "TRUE" } Add(in1 := 1, in2 := #Stanje, out => #Stanje)
   END_RUNG
   // the same network as SCL:
   IF (#Stanje = 0) AND "Ready_Flag" AND NOT "Lokacije_DB".L1_vhod_1.zasedenost THEN
       #Stanje := 1 + #Stanje;
   END_IF;
END_REGION

REGION Network 4: Stanje 0.1: Preverimo ali je material na vhodu in zgeneriramo vse potrebne podatke za recept.
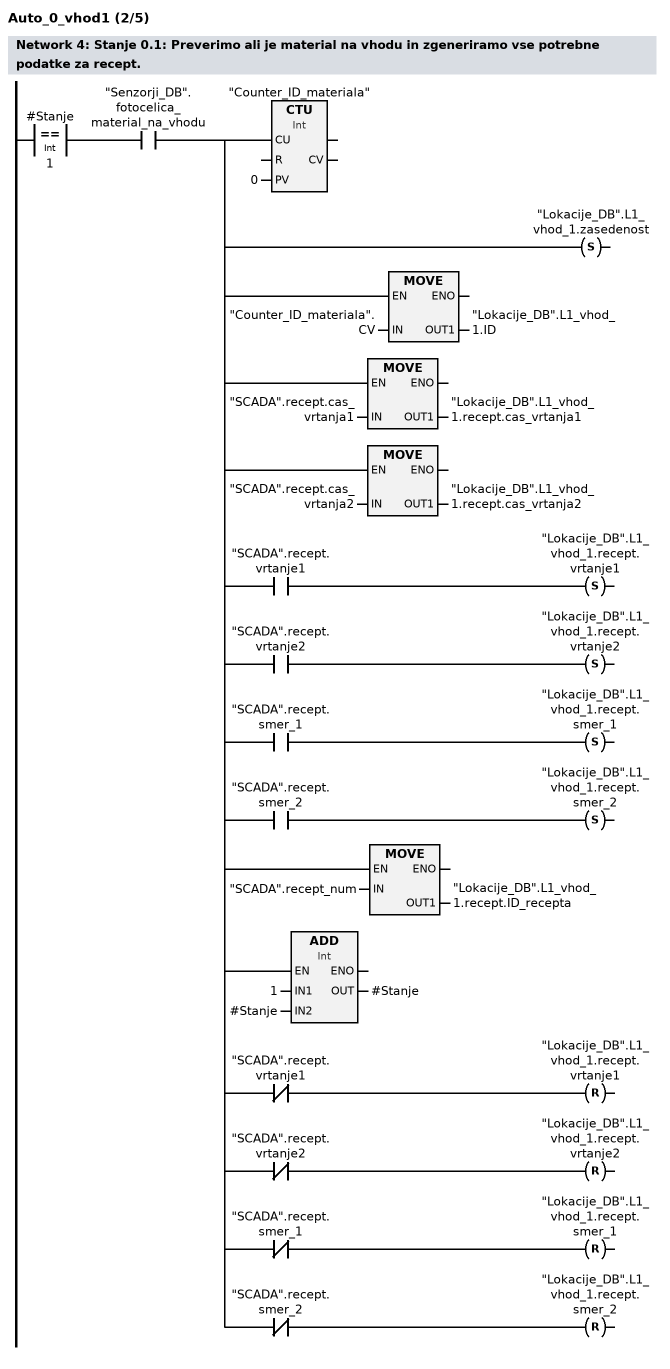
   #_w1 := (#Stanje = 1) AND "Senzorji_DB".fotocelica_material_na_vhodu;
   "Counter_ID_materiala".CTU(CU := #_w1, PV := 0);
   IF #_w1 THEN
       "Lokacije_DB".L1_vhod_1.zasedenost := TRUE;
       "Lokacije_DB".L1_vhod_1.ID := "Counter_ID_materiala".CV;
       "Lokacije_DB".L1_vhod_1.recept.cas_vrtanja1 := "SCADA".recept.cas_vrtanja1;
       "Lokacije_DB".L1_vhod_1.recept.cas_vrtanja2 := "SCADA".recept.cas_vrtanja2;
   END_IF;
   IF #_w1 AND "SCADA".recept.vrtanje1 THEN "Lokacije_DB".L1_vhod_1.recept.vrtanje1 := TRUE; END_IF;
   IF #_w1 AND "SCADA".recept.vrtanje2 THEN "Lokacije_DB".L1_vhod_1.recept.vrtanje2 := TRUE; END_IF;
   IF #_w1 AND "SCADA".recept.smer_1 THEN "Lokacije_DB".L1_vhod_1.recept.smer_1 := TRUE; END_IF;
   IF #_w1 AND "SCADA".recept.smer_2 THEN "Lokacije_DB".L1_vhod_1.recept.smer_2 := TRUE; END_IF;
   IF #_w1 THEN
       "Lokacije_DB".L1_vhod_1.recept.ID_recepta := "SCADA".recept_num;
       #Stanje := 1 + #Stanje;
   END_IF;
   IF #_w1 AND NOT "SCADA".recept.vrtanje1 THEN "Lokacije_DB".L1_vhod_1.recept.vrtanje1 := FALSE; END_IF;
   IF #_w1 AND NOT "SCADA".recept.vrtanje2 THEN "Lokacije_DB".L1_vhod_1.recept.vrtanje2 := FALSE; END_IF;
   IF #_w1 AND NOT "SCADA".recept.smer_1 THEN "Lokacije_DB".L1_vhod_1.recept.smer_1 := FALSE; END_IF;
   IF #_w1 AND NOT "SCADA".recept.smer_2 THEN "Lokacije_DB".L1_vhod_1.recept.smer_2 := FALSE; END_IF;
END_REGION

REGION Network 5: Stanje 0.2: Če druga fotocelica ni zasedena, premaknemo material naprej.
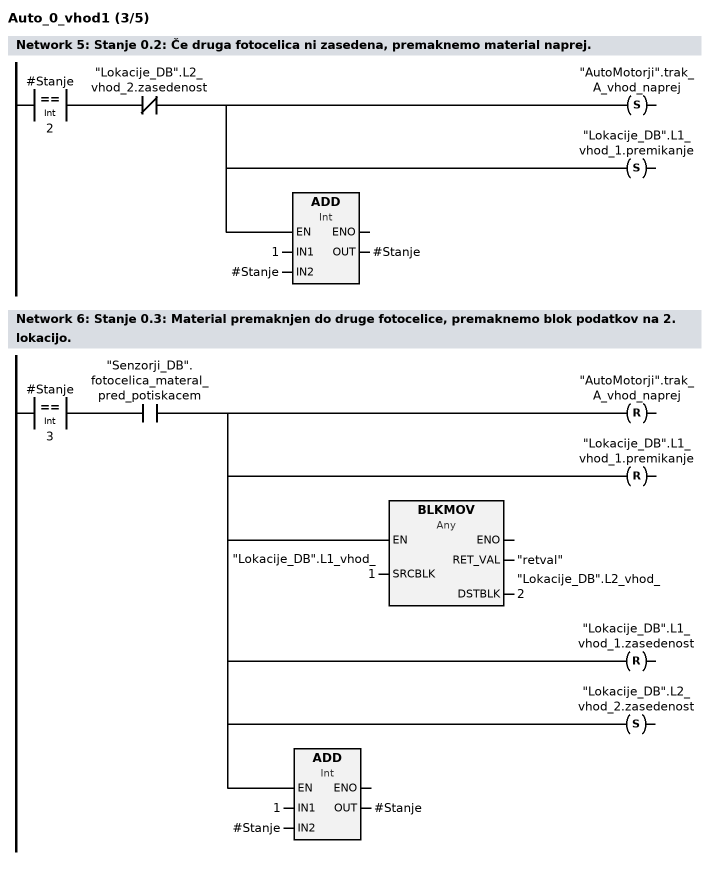
   RUNG wire#powerrail
      { S7_Templates := "SrcType := Int" } EQ_Contact(in1 := #Stanje, in2 := 2)
      I_Contact( "Lokacije_DB".L2_vhod_2.zasedenost )
      wire#w1
      S_Coil( "AutoMotorji".trak_A_vhod_naprej )
   END_RUNG
   RUNG wire#w1
      S_Coil( "Lokacije_DB".L1_vhod_1.premikanje )
   END_RUNG
   RUNG wire#w1
      { S7_Templates := "SrcType := Int"; S7_GenerateENO := "TRUE" } Add(in1 := 1, in2 := #Stanje, out => #Stanje)
   END_RUNG
   // the same network as SCL:
   IF (#Stanje = 2) AND NOT "Lokacije_DB".L2_vhod_2.zasedenost THEN
       "AutoMotorji".trak_A_vhod_naprej := TRUE;
       "Lokacije_DB".L1_vhod_1.premikanje := TRUE;
       #Stanje := 1 + #Stanje;
   END_IF;
END_REGION

REGION Network 6: Stanje 0.3: Material premaknjen do druge fotocelice, premaknemo blok podatkov na 2. lokacijo.
   IF (#Stanje = 3) AND "Senzorji_DB".fotocelica_materal_pred_potiskacem THEN
       "AutoMotorji".trak_A_vhod_naprej := FALSE;
       "Lokacije_DB".L1_vhod_1.premikanje := FALSE;
   END_IF;
   #_w1 := (#Stanje = 3) AND "Senzorji_DB".fotocelica_materal_pred_potiskacem;
   IF #_w1 THEN
       "retval" := BLKMOV(SRCBLK := "Lokacije_DB".L1_vhod_1, DSTBLK => "Lokacije_DB".L2_vhod_2);
       "Lokacije_DB".L1_vhod_1.zasedenost := FALSE;
       "Lokacije_DB".L2_vhod_2.zasedenost := TRUE;
       #Stanje := 1 + #Stanje;
   END_IF;
END_REGION

REGION Network 7: Stanje 0.4: Če potiskač ni zaseden, premaknemo material pred potiskač.
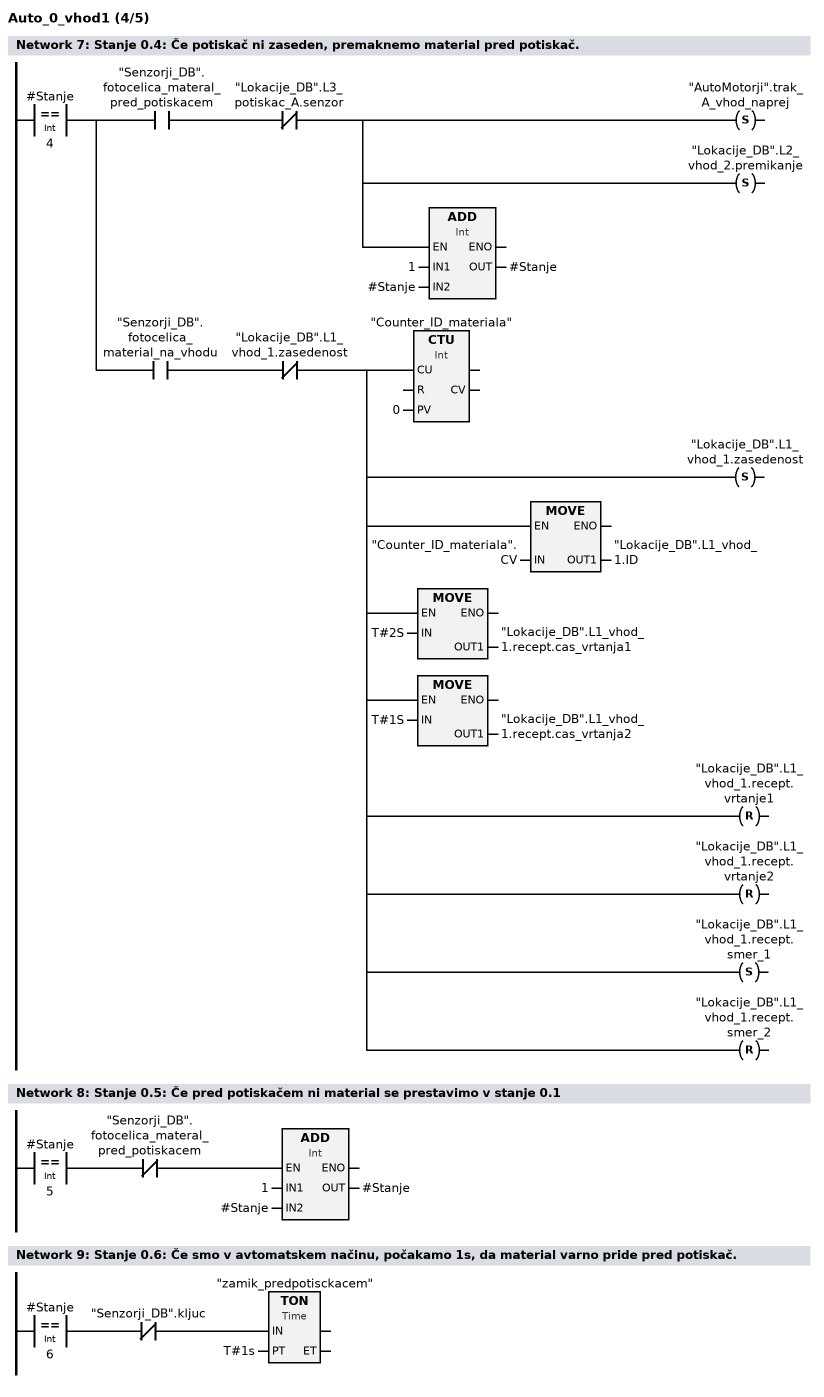
   #_w1 := #Stanje = 4;
   IF #_w1 AND "Senzorji_DB".fotocelica_materal_pred_potiskacem AND NOT "Lokacije_DB".L3_potiskac_A.senzor THEN
       "AutoMotorji".trak_A_vhod_naprej := TRUE;
       "Lokacije_DB".L2_vhod_2.premikanje := TRUE;
       #Stanje := 1 + #Stanje;
   END_IF;
   #_w2 := #_w1 AND "Senzorji_DB".fotocelica_material_na_vhodu AND NOT "Lokacije_DB".L1_vhod_1.zasedenost;
   "Counter_ID_materiala".CTU(CU := #_w2, PV := 0);
   IF #_w2 THEN
       "Lokacije_DB".L1_vhod_1.zasedenost := TRUE;
       "Lokacije_DB".L1_vhod_1.ID := "Counter_ID_materiala".CV;
       "Lokacije_DB".L1_vhod_1.recept.cas_vrtanja1 := T#2S;
       "Lokacije_DB".L1_vhod_1.recept.cas_vrtanja2 := T#1S;
       "Lokacije_DB".L1_vhod_1.recept.vrtanje1 := FALSE;
       "Lokacije_DB".L1_vhod_1.recept.vrtanje2 := FALSE;
       "Lokacije_DB".L1_vhod_1.recept.smer_1 := TRUE;
       "Lokacije_DB".L1_vhod_1.recept.smer_2 := FALSE;
   END_IF;
END_REGION

REGION Network 8: Stanje 0.5: Če pred potiskačem ni material se prestavimo v stanje 0.1
   RUNG wire#powerrail
      { S7_Templates := "SrcType := Int" } EQ_Contact(in1 := #Stanje, in2 := 5)
      I_Contact( "Senzorji_DB".fotocelica_materal_pred_potiskacem )
      { S7_Templates := "SrcType := Int"; S7_GenerateENO := "TRUE" } Add(in1 := 1, in2 := #Stanje, out => #Stanje)
   END_RUNG
   // the same network as SCL:
   IF (#Stanje = 5) AND NOT "Senzorji_DB".fotocelica_materal_pred_potiskacem THEN
       #Stanje := 1 + #Stanje;
   END_IF;
END_REGION

REGION Network 9: Stanje 0.6: Če smo v avtomatskem načinu, počakamo 1s, da material varno pride pred potiskač.
   "zamik_predpotisckacem".TON(IN := (#Stanje = 6) AND NOT "Senzorji_DB".kljuc, PT := T#1s);
END_REGION

REGION Network 10: Stanje0.6: Premaknemo blok podatkov na 3. lokacijo in gremo v stanje 0.0.
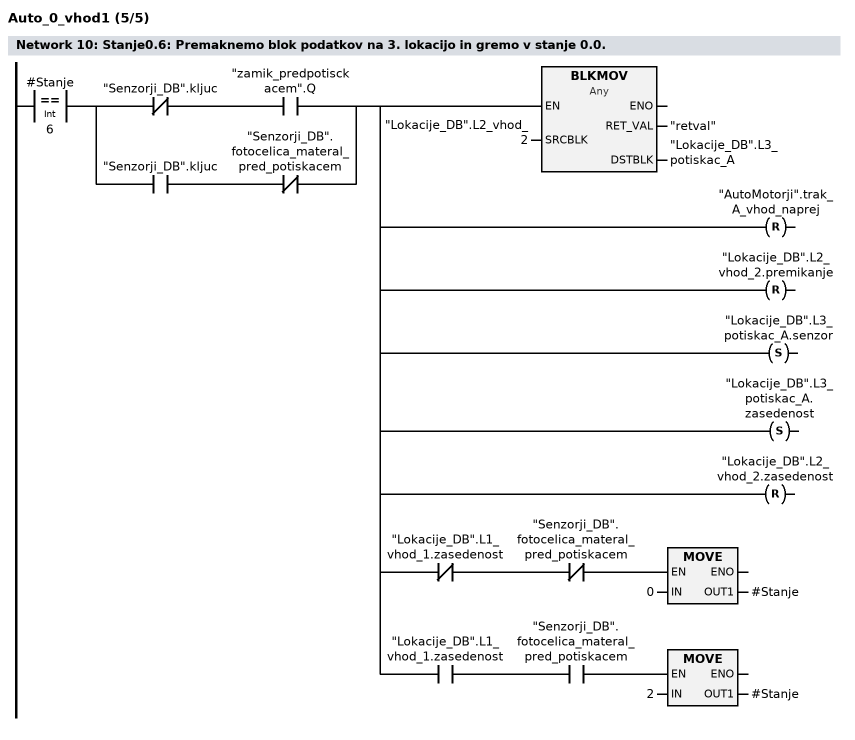
   #_w1 := (#Stanje = 6) AND ((NOT "Senzorji_DB".kljuc AND "zamik_predpotisckacem".Q) OR ("Senzorji_DB".kljuc AND NOT "Senzorji_DB".fotocelica_materal_pred_potiskacem));
   IF #_w1 THEN
       "retval" := BLKMOV(SRCBLK := "Lokacije_DB".L2_vhod_2, DSTBLK => "Lokacije_DB".L3_potiskac_A);
       "AutoMotorji".trak_A_vhod_naprej := FALSE;
       "Lokacije_DB".L2_vhod_2.premikanje := FALSE;
       "Lokacije_DB".L3_potiskac_A.senzor := TRUE;
       "Lokacije_DB".L3_potiskac_A.zasedenost := TRUE;
       "Lokacije_DB".L2_vhod_2.zasedenost := FALSE;
   END_IF;
   IF #_w1 AND NOT "Lokacije_DB".L1_vhod_1.zasedenost AND NOT "Senzorji_DB".fotocelica_materal_pred_potiskacem THEN
       #Stanje := 0;
   END_IF;
   IF #_w1 AND "Lokacije_DB".L1_vhod_1.zasedenost AND "Senzorji_DB".fotocelica_materal_pred_potiskacem THEN
       #Stanje := 2;
   END_IF;
END_REGION
END_FUNCTION_BLOCK

FUNCTION_BLOCK "Auto_3_B_Naprava"   // FB7, LAD
TITLE = Stanje 3: B naprava
{ S7_Optimized_Access := 'FALSE' }
VERSION : 0.1
// Vrtanje z B napravo in premik materiala pred potiskač B.
   VAR_TEMP   // added for the SCL form of the ladder/FBD networks
      _w1 : Bool;
      _w2 : Bool;
      _w3 : Bool;
      _w4 : Bool;
      _w5 : Bool;
   END_VAR
BEGIN

REGION Network 1
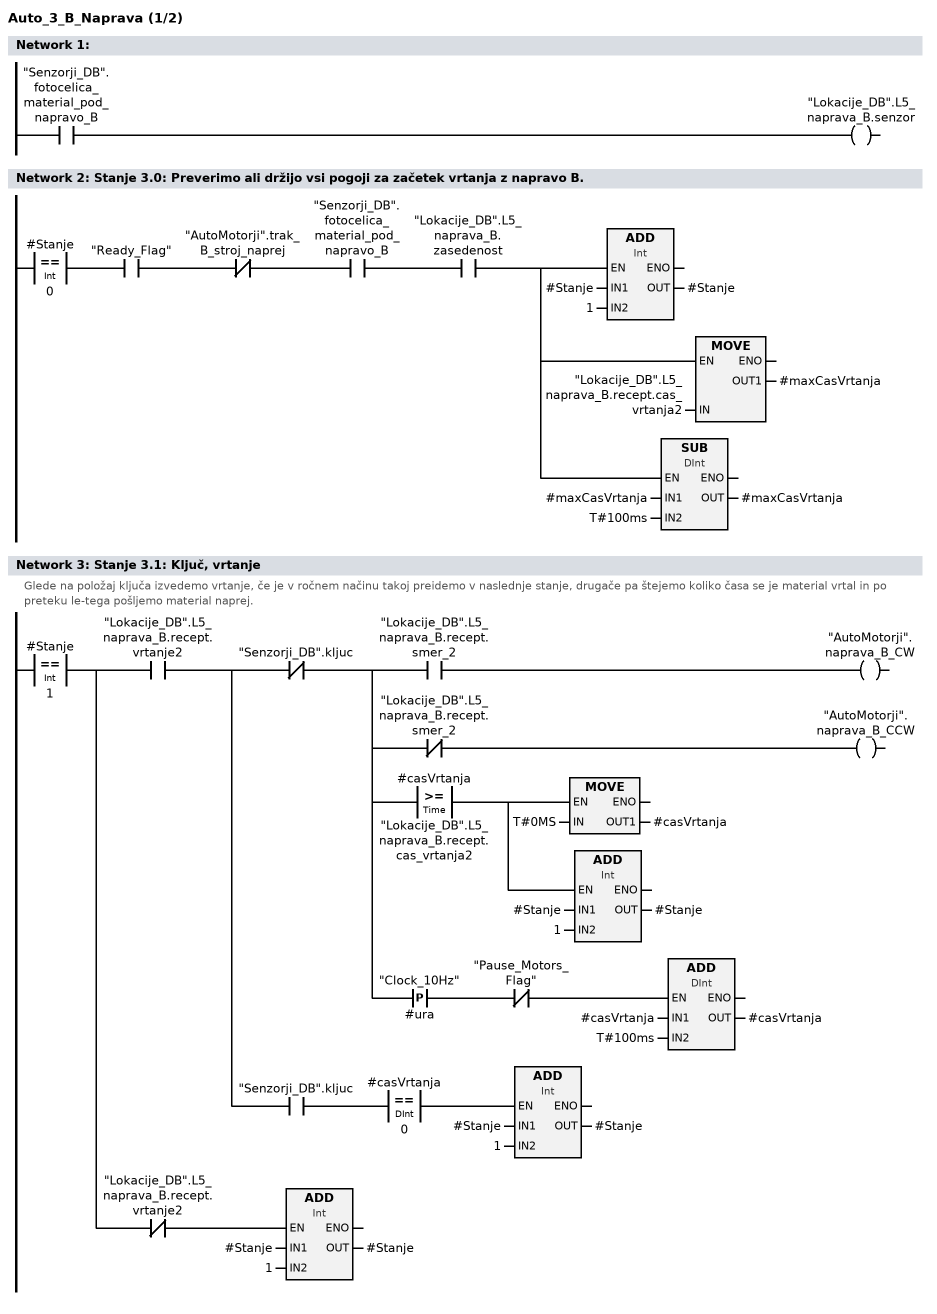
   RUNG wire#powerrail
      Contact( "Senzorji_DB".fotocelica_material_pod_napravo_B )
      Coil( "Lokacije_DB".L5_naprava_B.senzor )
   END_RUNG
   // the same network as SCL:
   "Lokacije_DB".L5_naprava_B.senzor := "Senzorji_DB".fotocelica_material_pod_napravo_B;
END_REGION

REGION Network 2: Stanje 3.0: Preverimo ali držijo vsi pogoji za začetek vrtanja z napravo B.
   RUNG wire#powerrail
      { S7_Templates := "SrcType := Int" } EQ_Contact(in1 := #Stanje, in2 := 0)
      Contact( "Ready_Flag" )
      I_Contact( "AutoMotorji".trak_B_stroj_naprej )
      Contact( "Senzorji_DB".fotocelica_material_pod_napravo_B )
      Contact( "Lokacije_DB".L5_naprava_B.zasedenost )
      wire#w1
      { S7_Templates := "SrcType := Int"; S7_GenerateENO := "TRUE" } Add(in1 := #Stanje, in2 := 1, out => #Stanje)
   END_RUNG
   RUNG wire#w1
      { S7_GenerateENO := "TRUE" } Move(in := "Lokacije_DB".L5_naprava_B.recept.cas_vrtanja2, out1 => #maxCasVrtanja)
   END_RUNG
   RUNG wire#w1
      { S7_Templates := "SrcType := DInt"; S7_GenerateENO := "TRUE" } Sub(in1 := #maxCasVrtanja, in2 := T#100ms, out => #maxCasVrtanja)
   END_RUNG
   // the same network as SCL:
   #_w1 := (#Stanje = 0) AND "Ready_Flag" AND NOT "AutoMotorji".trak_B_stroj_naprej AND "Senzorji_DB".fotocelica_material_pod_napravo_B AND "Lokacije_DB".L5_naprava_B.zasedenost;
   IF #_w1 THEN
       #Stanje := #Stanje + 1;
       #maxCasVrtanja := "Lokacije_DB".L5_naprava_B.recept.cas_vrtanja2;
       #maxCasVrtanja := #maxCasVrtanja - T#100ms;
   END_IF;
END_REGION

REGION Network 3: Stanje 3.1: Ključ, vrtanje
   // Glede na položaj ključa izvedemo vrtanje, če je v ročnem načinu takoj preidemo v naslednje stanje, drugače pa štejemo koliko časa se je material vrtal in po preteku le-tega pošljemo material naprej.
   RUNG wire#powerrail
      { S7_Templates := "SrcType := Int" } EQ_Contact(in1 := #Stanje, in2 := 1)
      wire#w1
      Contact( "Lokacije_DB".L5_naprava_B.recept.vrtanje2 )
      wire#w2
      I_Contact( "Senzorji_DB".kljuc )
      wire#w3
      Contact( "Lokacije_DB".L5_naprava_B.recept.smer_2 )
      Coil( "AutoMotorji".naprava_B_CW )
   END_RUNG
   RUNG wire#w3
      I_Contact( "Lokacije_DB".L5_naprava_B.recept.smer_2 )
      Coil( "AutoMotorji".naprava_B_CCW )
   END_RUNG
   RUNG wire#w3
      { S7_Templates := "SrcType := Time" } GE_Contact(in1 := #casVrtanja, in2 := "Lokacije_DB".L5_naprava_B.recept.cas_vrtanja2)
      wire#w4
      { S7_GenerateENO := "TRUE" } Move(in := T#0MS, out1 => #casVrtanja)
   END_RUNG
   RUNG wire#w4
      { S7_Templates := "SrcType := Int"; S7_GenerateENO := "TRUE" } Add(in1 := #Stanje, in2 := 1, out => #Stanje)
   END_RUNG
   RUNG wire#w3
      P_Contact(operand := "Clock_10Hz", bit := #ura)
      I_Contact( "Pause_Motors_Flag" )
      { S7_Templates := "SrcType := DInt"; S7_GenerateENO := "TRUE" } Add(in1 := #casVrtanja, in2 := T#100ms, out => #casVrtanja)
   END_RUNG
   RUNG wire#w2
      Contact( "Senzorji_DB".kljuc )
      { S7_Templates := "SrcType := DInt" } EQ_Contact(in1 := #casVrtanja, in2 := 0)
      { S7_Templates := "SrcType := Int"; S7_GenerateENO := "TRUE" } Add(in1 := #Stanje, in2 := 1, out => #Stanje)
   END_RUNG
   RUNG wire#w1
      I_Contact( "Lokacije_DB".L5_naprava_B.recept.vrtanje2 )
      { S7_Templates := "SrcType := Int"; S7_GenerateENO := "TRUE" } Add(in1 := #Stanje, in2 := 1, out => #Stanje)
   END_RUNG
   // the same network as SCL:
   #_w1 := #Stanje = 1;
   #_w2 := #_w1 AND "Lokacije_DB".L5_naprava_B.recept.vrtanje2;
   #_w3 := #_w2 AND NOT "Senzorji_DB".kljuc;
   "AutoMotorji".naprava_B_CW := #_w3 AND "Lokacije_DB".L5_naprava_B.recept.smer_2;
   "AutoMotorji".naprava_B_CCW := #_w3 AND NOT "Lokacije_DB".L5_naprava_B.recept.smer_2;
   #_w4 := #_w3 AND (#casVrtanja >= "Lokacije_DB".L5_naprava_B.recept.cas_vrtanja2);
   IF #_w4 THEN
       #casVrtanja := T#0MS;
       #Stanje := #Stanje + 1;
   END_IF;
   #_w5 := #_w3 AND "Clock_10Hz" AND NOT #ura;   // rising edge of "Clock_10Hz"
   #ura := "Clock_10Hz";
   IF #_w5 AND NOT "Pause_Motors_Flag" THEN #casVrtanja := #casVrtanja + T#100ms; END_IF;
   IF #_w2 AND "Senzorji_DB".kljuc AND (#casVrtanja = 0) THEN #Stanje := #Stanje + 1; END_IF;
   IF #_w1 AND NOT "Lokacije_DB".L5_naprava_B.recept.vrtanje2 THEN #Stanje := #Stanje + 1; END_IF;
END_REGION

REGION Network 4: Stanje 3.2: Začnemo premikati trak pod napravo B.
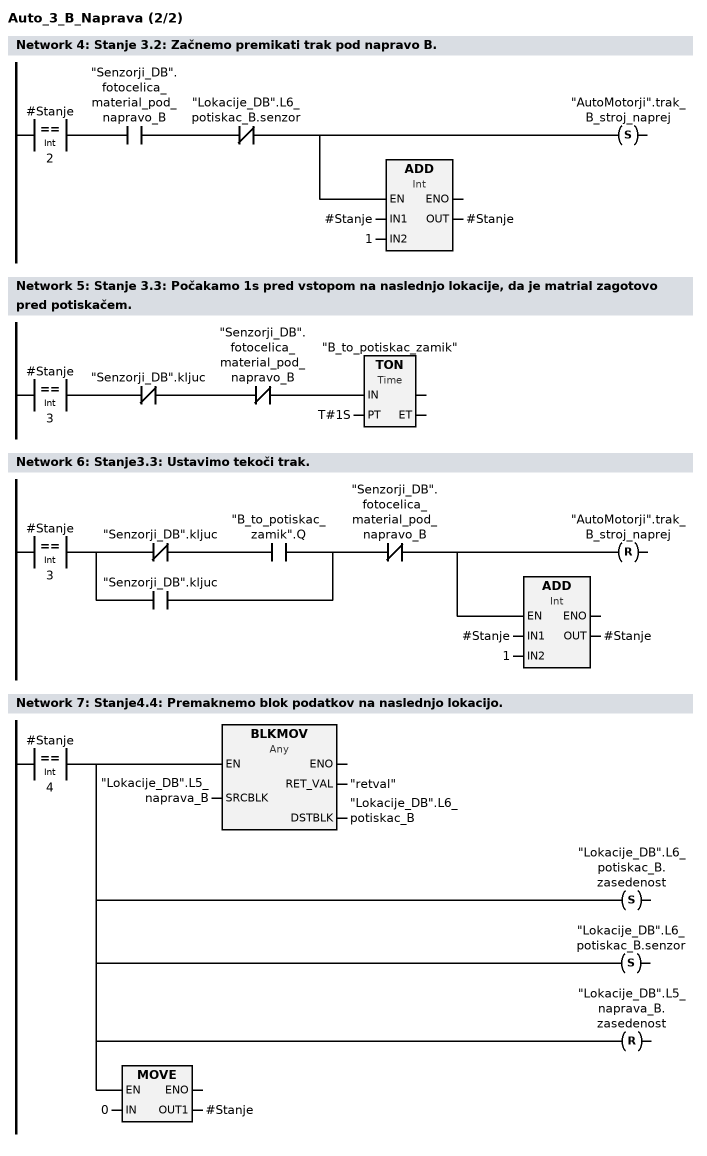
   RUNG wire#powerrail
      { S7_Templates := "SrcType := Int" } EQ_Contact(in1 := #Stanje, in2 := 2)
      Contact( "Senzorji_DB".fotocelica_material_pod_napravo_B )
      I_Contact( "Lokacije_DB".L6_potiskac_B.senzor )
      wire#w1
      S_Coil( "AutoMotorji".trak_B_stroj_naprej )
   END_RUNG
   RUNG wire#w1
      { S7_Templates := "SrcType := Int"; S7_GenerateENO := "TRUE" } Add(in1 := #Stanje, in2 := 1, out => #Stanje)
   END_RUNG
   // the same network as SCL:
   IF (#Stanje = 2) AND "Senzorji_DB".fotocelica_material_pod_napravo_B AND NOT "Lokacije_DB".L6_potiskac_B.senzor THEN
       "AutoMotorji".trak_B_stroj_naprej := TRUE;
       #Stanje := #Stanje + 1;
   END_IF;
END_REGION

REGION Network 5: Stanje 3.3: Počakamo 1s pred vstopom na naslednjo lokacije, da je matrial zagotovo pred potiskačem.
   "B_to_potiskac_zamik".TON(IN := (#Stanje = 3) AND NOT "Senzorji_DB".kljuc AND NOT "Senzorji_DB".fotocelica_material_pod_napravo_B,
                           PT := T#1S);
END_REGION

REGION Network 6: Stanje3.3: Ustavimo tekoči trak.
   RUNG wire#powerrail
      { S7_Templates := "SrcType := Int" } EQ_Contact(in1 := #Stanje, in2 := 3)
      wire#w1
      I_Contact( "Senzorji_DB".kljuc )
      Contact( "B_to_potiskac_zamik".Q )
      wire#w2
      I_Contact( "Senzorji_DB".fotocelica_material_pod_napravo_B )
      wire#w3
      R_Coil( "AutoMotorji".trak_B_stroj_naprej )
   END_RUNG
   RUNG wire#w1
      Contact( "Senzorji_DB".kljuc )
   END_RUNG wire#w2
   RUNG wire#w3
      { S7_Templates := "SrcType := Int"; S7_GenerateENO := "TRUE" } Add(in1 := #Stanje, in2 := 1, out => #Stanje)
   END_RUNG
   // the same network as SCL:
   IF (#Stanje = 3) AND ((NOT "Senzorji_DB".kljuc AND "B_to_potiskac_zamik".Q) OR "Senzorji_DB".kljuc) AND NOT "Senzorji_DB".fotocelica_material_pod_napravo_B THEN
       "AutoMotorji".trak_B_stroj_naprej := FALSE;
       #Stanje := #Stanje + 1;
   END_IF;
END_REGION

REGION Network 7: Stanje4.4: Premaknemo blok podatkov na naslednjo lokacijo.
   IF #Stanje = 4 THEN
       "retval" := BLKMOV(SRCBLK := "Lokacije_DB".L5_naprava_B, DSTBLK => "Lokacije_DB".L6_potiskac_B);
       "Lokacije_DB".L6_potiskac_B.zasedenost := TRUE;
       "Lokacije_DB".L6_potiskac_B.senzor := TRUE;
       "Lokacije_DB".L5_naprava_B.zasedenost := FALSE;
       #Stanje := 0;
   END_IF;
END_REGION
END_FUNCTION_BLOCK

FUNCTION_BLOCK "Auto_4_Potiskac"   // FB8, LAD
TITLE = Stanje 4: Potiskač B
{ S7_Optimized_Access := 'FALSE' }
VERSION : 0.1
// Premikanje potiskača B, da spravi material s tekočega traku pod napravo B do tekočega traku na izhodu.
   VAR_TEMP   // added for the SCL form of the ladder/FBD networks
      _w1 : Bool;
      _w2 : Bool;
      _w3 : Bool;
      _w4 : Bool;
   END_VAR
BEGIN

REGION Network 1: Stanje 4.0: Preverimo ali držijo vsi pogoji za začetek premikanja potiskača B.
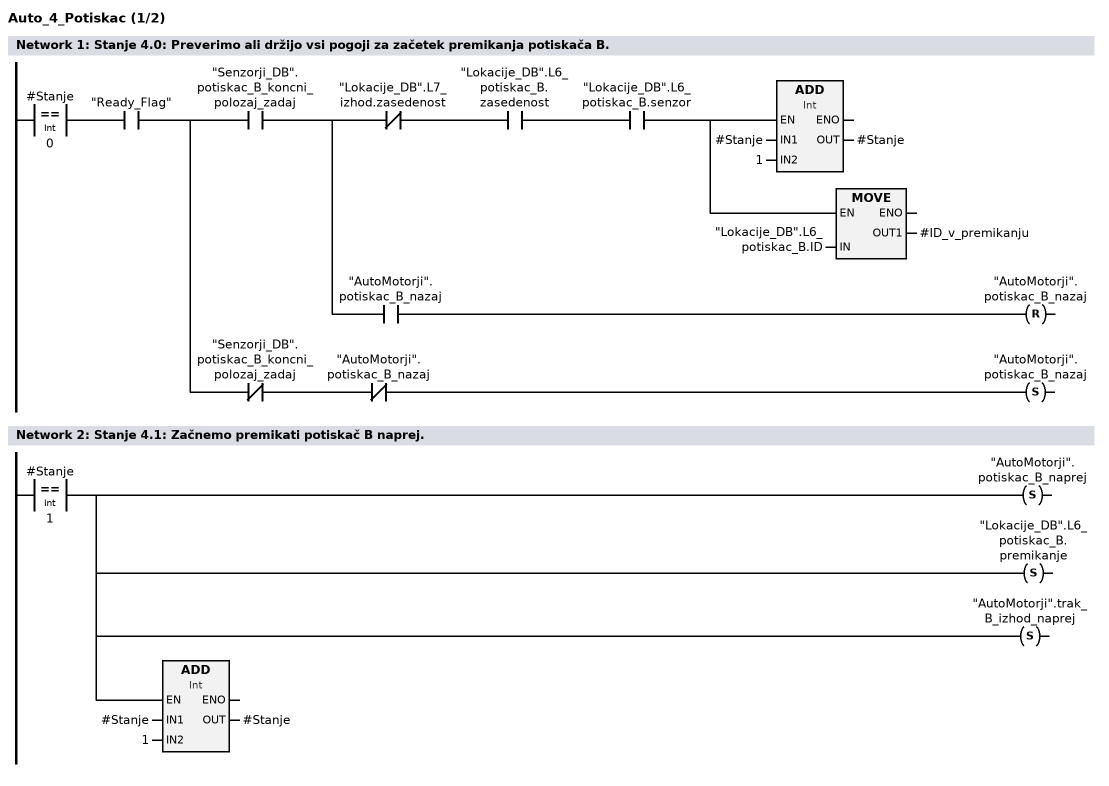
   RUNG wire#powerrail
      { S7_Templates := "SrcType := Int" } EQ_Contact(in1 := #Stanje, in2 := 0)
      Contact( "Ready_Flag" )
      wire#w1
      Contact( "Senzorji_DB".potiskac_B_koncni_polozaj_zadaj )
      wire#w2
      I_Contact( "Lokacije_DB".L7_izhod.zasedenost )
      Contact( "Lokacije_DB".L6_potiskac_B.zasedenost )
      Contact( "Lokacije_DB".L6_potiskac_B.senzor )
      wire#w3
      { S7_Templates := "SrcType := Int"; S7_GenerateENO := "TRUE" } Add(in1 := #Stanje, in2 := 1, out => #Stanje)
   END_RUNG
   RUNG wire#w3
      { S7_GenerateENO := "TRUE" } Move(in := "Lokacije_DB".L6_potiskac_B.ID, out1 => #ID_v_premikanju)
   END_RUNG
   RUNG wire#w2
      Contact( "AutoMotorji".potiskac_B_nazaj )
      R_Coil( "AutoMotorji".potiskac_B_nazaj )
   END_RUNG
   RUNG wire#w1
      I_Contact( "Senzorji_DB".potiskac_B_koncni_polozaj_zadaj )
      I_Contact( "AutoMotorji".potiskac_B_nazaj )
      S_Coil( "AutoMotorji".potiskac_B_nazaj )
   END_RUNG
   // the same network as SCL:
   #_w1 := (#Stanje = 0) AND "Ready_Flag";
   #_w2 := #_w1 AND "Senzorji_DB".potiskac_B_koncni_polozaj_zadaj;
   IF #_w2 AND NOT "Lokacije_DB".L7_izhod.zasedenost AND "Lokacije_DB".L6_potiskac_B.zasedenost AND "Lokacije_DB".L6_potiskac_B.senzor THEN
       #Stanje := #Stanje + 1;
       #ID_v_premikanju := "Lokacije_DB".L6_potiskac_B.ID;
   END_IF;
   IF #_w2 AND "AutoMotorji".potiskac_B_nazaj THEN "AutoMotorji".potiskac_B_nazaj := FALSE; END_IF;
   IF #_w1 AND NOT "Senzorji_DB".potiskac_B_koncni_polozaj_zadaj AND NOT "AutoMotorji".potiskac_B_nazaj THEN
       "AutoMotorji".potiskac_B_nazaj := TRUE;
   END_IF;
END_REGION

REGION Network 2: Stanje 4.1: Začnemo premikati potiskač B naprej.
   RUNG wire#powerrail
      { S7_Templates := "SrcType := Int" } EQ_Contact(in1 := #Stanje, in2 := 1)
      wire#w1
      S_Coil( "AutoMotorji".potiskac_B_naprej )
   END_RUNG
   RUNG wire#w1
      S_Coil( "Lokacije_DB".L6_potiskac_B.premikanje )
   END_RUNG
   RUNG wire#w1
      S_Coil( "AutoMotorji".trak_B_izhod_naprej )
   END_RUNG
   RUNG wire#w1
      { S7_Templates := "SrcType := Int"; S7_GenerateENO := "TRUE" } Add(in1 := #Stanje, in2 := 1, out => #Stanje)
   END_RUNG
   // the same network as SCL:
   IF #Stanje = 1 THEN
       "AutoMotorji".potiskac_B_naprej := TRUE;
       "Lokacije_DB".L6_potiskac_B.premikanje := TRUE;
       "AutoMotorji".trak_B_izhod_naprej := TRUE;
       #Stanje := #Stanje + 1;
   END_IF;
END_REGION

REGION Network 3: Stanje 4.2: Potiskač naprej, fotocelica, potiskač nazaj.
   // Premikamo potiskač naprej do končnega položaj, ko pride material do fotocelice, vrtimo potiskač nazaj do končnega položaja.
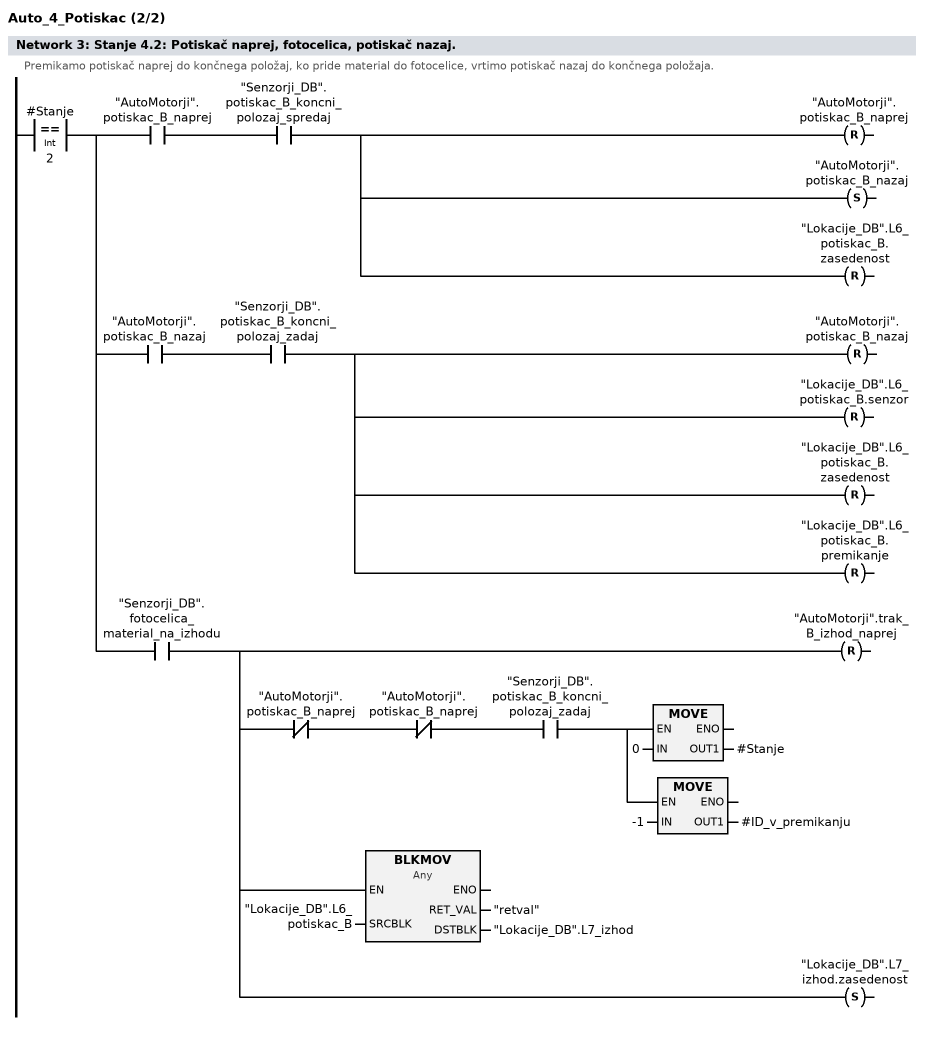
   #_w1 := #Stanje = 2;
   #_w2 := #_w1 AND "AutoMotorji".potiskac_B_naprej AND "Senzorji_DB".potiskac_B_koncni_polozaj_spredaj;
   IF #_w2 THEN
       "AutoMotorji".potiskac_B_naprej := FALSE;
       "AutoMotorji".potiskac_B_nazaj := TRUE;
       "Lokacije_DB".L6_potiskac_B.zasedenost := FALSE;
   END_IF;
   #_w3 := #_w1 AND "AutoMotorji".potiskac_B_nazaj AND "Senzorji_DB".potiskac_B_koncni_polozaj_zadaj;
   IF #_w3 THEN
       "AutoMotorji".potiskac_B_nazaj := FALSE;
       "Lokacije_DB".L6_potiskac_B.senzor := FALSE;
       "Lokacije_DB".L6_potiskac_B.zasedenost := FALSE;
       "Lokacije_DB".L6_potiskac_B.premikanje := FALSE;
   END_IF;
   #_w4 := #_w1 AND "Senzorji_DB".fotocelica_material_na_izhodu;
   IF #_w4 THEN "AutoMotorji".trak_B_izhod_naprej := FALSE; END_IF;
   IF #_w4 AND NOT "AutoMotorji".potiskac_B_naprej AND NOT "AutoMotorji".potiskac_B_naprej AND "Senzorji_DB".potiskac_B_koncni_polozaj_zadaj THEN
       #Stanje := 0;
       #ID_v_premikanju := -1;
   END_IF;
   IF #_w4 THEN
       "retval" := BLKMOV(SRCBLK := "Lokacije_DB".L6_potiskac_B, DSTBLK => "Lokacije_DB".L7_izhod);
       "Lokacije_DB".L7_izhod.zasedenost := TRUE;
   END_IF;
END_REGION
END_FUNCTION_BLOCK

FUNCTION_BLOCK "Auto_5_Izhod"   // FB9, LAD
TITLE = Stanje 5: Izhodni tekoči trak.
{ S7_Optimized_Access := 'FALSE' }
VERSION : 0.1
// Transport materiala do konca procesne linije.
   VAR_TEMP   // added for the SCL form of the ladder/FBD networks
      _w1 : Bool;
   END_VAR
BEGIN

REGION Network 1
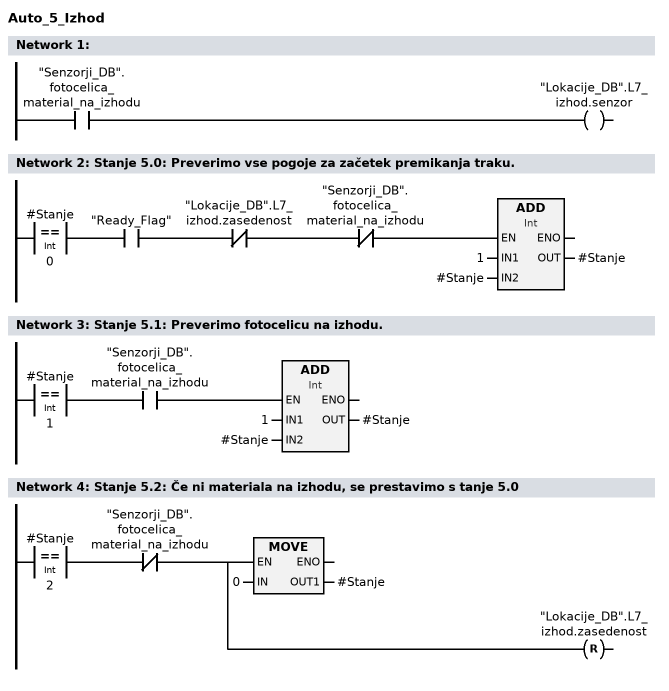
   RUNG wire#powerrail
      Contact( "Senzorji_DB".fotocelica_material_na_izhodu )
      Coil( "Lokacije_DB".L7_izhod.senzor )
   END_RUNG
   // the same network as SCL:
   "Lokacije_DB".L7_izhod.senzor := "Senzorji_DB".fotocelica_material_na_izhodu;
END_REGION

REGION Network 2: Stanje 5.0: Preverimo vse pogoje za začetek premikanja traku.
   RUNG wire#powerrail
      { S7_Templates := "SrcType := Int" } EQ_Contact(in1 := #Stanje, in2 := 0)
      Contact( "Ready_Flag" )
      I_Contact( "Lokacije_DB".L7_izhod.zasedenost )
      I_Contact( "Senzorji_DB".fotocelica_material_na_izhodu )
      { S7_Templates := "SrcType := Int"; S7_GenerateENO := "TRUE" } Add(in1 := 1, in2 := #Stanje, out => #Stanje)
   END_RUNG
   // the same network as SCL:
   IF (#Stanje = 0) AND "Ready_Flag" AND NOT "Lokacije_DB".L7_izhod.zasedenost AND NOT "Senzorji_DB".fotocelica_material_na_izhodu THEN
       #Stanje := 1 + #Stanje;
   END_IF;
END_REGION

REGION Network 3: Stanje 5.1: Preverimo fotocelicu na izhodu.
   RUNG wire#powerrail
      { S7_Templates := "SrcType := Int" } EQ_Contact(in1 := #Stanje, in2 := 1)
      Contact( "Senzorji_DB".fotocelica_material_na_izhodu )
      { S7_Templates := "SrcType := Int"; S7_GenerateENO := "TRUE" } Add(in1 := 1, in2 := #Stanje, out => #Stanje)
   END_RUNG
   // the same network as SCL:
   IF (#Stanje = 1) AND "Senzorji_DB".fotocelica_material_na_izhodu THEN #Stanje := 1 + #Stanje; END_IF;
END_REGION

REGION Network 4: Stanje 5.2: Če ni materiala na izhodu, se prestavimo s tanje 5.0
   RUNG wire#powerrail
      { S7_Templates := "SrcType := Int" } EQ_Contact(in1 := #Stanje, in2 := 2)
      I_Contact( "Senzorji_DB".fotocelica_material_na_izhodu )
      wire#w1
      { S7_GenerateENO := "TRUE" } Move(in := 0, out1 => #Stanje)
   END_RUNG
   RUNG wire#w1
      R_Coil( "Lokacije_DB".L7_izhod.zasedenost )
   END_RUNG
   // the same network as SCL:
   #_w1 := (#Stanje = 2) AND NOT "Senzorji_DB".fotocelica_material_na_izhodu;
   IF #_w1 THEN
       #Stanje := 0;
       "Lokacije_DB".L7_izhod.zasedenost := FALSE;
   END_IF;
END_REGION
END_FUNCTION_BLOCK

// folder: GlavniProgram/Alarmi

FUNCTION_BLOCK "Alarmi"   // FB10, SCL
{ S7_Optimized_Access := 'FALSE' }
VERSION : 0.1
BEGIN



   IF "Startup_Flag" THEN


       IF "Senzorji_DB".fotocelica_material_na_vhodu OR "Senzorji_DB".fotocelica_materal_pred_potiskacem OR "Senzorji_DB".fotocelica_material_pod_napravo_A OR "Senzorji_DB".fotocelica_material_pod_napravo_B OR "Senzorji_DB".fotocelica_material_na_izhodu
           OR NOT ("Senzorji_DB".potiskac_A_koncni_polozaj_zadaj AND "Senzorji_DB".potiskac_B_koncni_polozaj_zadaj) THEN


               "SCADA".alarmi[14] := 1;
               "Pause_Motors_Flag" := 1;
       ELSE
           "Startup_Flag" := 0;
           "Ready_Flag" := 1;
           "Pause_Motors_Flag" := 0;

       END_IF;

   END_IF;

   IF NOT "Senzorji_DB".kljuc AND "Senzorji_DB".zelena_tipka THEN
       //POTRDITEV



       //"Pause_Motors_Flag" := 0
       ;

   END_IF;

   IF "Lokacije_DB".L1_vhod_1.zasedenost AND "Lokacije_DB".L2_vhod_2.zasedenost AND "Lokacije_DB".L3_potiskac_A.zasedenost AND "Lokacije_DB".L4_naprava_A.zasedenost AND "Lokacije_DB".L5_naprava_B.zasedenost AND "Lokacije_DB".L6_potiskac_B.zasedenost AND "Lokacije_DB".L7_izhod.zasedenost THEN
       // LINIJA JE POLNA ALARM15
       "SCADA".alarmi[15] := 1;
   END_IF;

   IF NOT "Senzorji_DB".kljuc AND NOT "Lokacije_DB".L1_vhod_1.zasedenost AND "Lokacije_DB".L2_vhod_2.senzor AND NOT "Lokacije_DB".L2_vhod_2.zasedenost THEN
       "SCADA".alarmi[0] := 1;
       "Pause_Motors_Flag" := 1;
       ;
   END_IF;

   IF NOT "Senzorji_DB".kljuc AND NOT "Lokacije_DB".L3_potiskac_A.zasedenost AND "Lokacije_DB".L4_naprava_A.senzor AND NOT "Lokacije_DB".L4_naprava_A.zasedenost THEN
       "SCADA".alarmi[1] := 1;
       "Pause_Motors_Flag" := 1;
       ;
   END_IF;

   IF NOT "Senzorji_DB".kljuc AND NOT "Lokacije_DB".L4_naprava_A.zasedenost AND "Lokacije_DB".L5_naprava_B.senzor AND NOT "Lokacije_DB".L5_naprava_B.zasedenost THEN
       "SCADA".alarmi[2] := 1;
       "Pause_Motors_Flag" := 1;
       ;
   END_IF;

   IF NOT "Senzorji_DB".kljuc AND NOT "Lokacije_DB".L6_potiskac_B.zasedenost AND "Lokacije_DB".L7_izhod.senzor AND NOT "Lokacije_DB".L7_izhod.zasedenost THEN
       "Pause_Motors_Flag" := 1;
       "SCADA".alarmi[3] := 1;
       ;
   END_IF;

   "L1_L2_Prehod0".TON(IN := NOT "Pause_Motors_Flag" AND NOT #l1_l2 AND "AutoMotorji".trak_A_vhod_naprej AND "Auto_0_vhod1_DB".Stanje = 3 AND NOT "Senzorji_DB".kljuc,
                       PT := T#3s,
                       Q => #l1_l2);
   IF #l1_l2 THEN
       "SCADA".alarmi[4] := 1;
       "Pause_Motors_Flag" := 1;


       ;
   END_IF;

   "L2_L4_Prehod".TON(IN :=  NOT "Pause_Motors_Flag" AND NOT #l3_l4 AND "AutoMotorji".trak_A_stroj_naprej AND "Auto_1_Potiskac_DB".Stanje = 2 AND NOT "Senzorji_DB".kljuc,
                      PT := T#5s,
                      Q => #l3_l4);
   IF #l3_l4 AND "Senzorji_DB".potiskac_A_koncni_polozaj_zadaj THEN //pocakamo da je potiskac noter da ni problemov 
       "SCADA".alarmi[5] := 1;
       "Pause_Motors_Flag" := 1;
   END_IF;

   "L4_L5".TON(IN := NOT "Pause_Motors_Flag" AND NOT #l4_l5 AND "AutoMotorji".trak_A_stroj_naprej AND "AutoMotorji".trak_B_stroj_naprej AND "Auto_2_A_Naprava_DB".Stanje = 3 AND NOT "Senzorji_DB".kljuc,
               PT := T#5s,
               Q => #l4_l5);

   IF #l4_l5 THEN
       "SCADA".alarmi[6] := 1;
       "Pause_Motors_Flag" := 1;
   END_IF;

   "L5_L7_Prehod".TON(IN :=  NOT "Pause_Motors_Flag" AND NOT #l6_l7 AND "AutoMotorji".trak_B_izhod_naprej AND "Auto_4_Potiskac_DB".Stanje = 2 AND NOT "Senzorji_DB".kljuc ,
                      PT := T#7s,
                      Q => #l6_l7);
   IF #l6_l7 AND "Senzorji_DB".potiskac_B_koncni_polozaj_zadaj THEN
       "SCADA".alarmi[7] := 1;
       "Pause_Motors_Flag" := 1;
   END_IF;

   IF "SCADA".recept_num <> #star_recept  THEN
       // Sprememba recepta
       "SCADA".alarmi[8] := 1;
       ;
   END_IF;
   #star_recept := "SCADA".recept_num;

   IF ("Senzorji_DB".kljuc = 1 AND #staro_kljuc = 0) OR ("Senzorji_DB".kljuc = 0 AND #staro_kljuc = 1) THEN
       // Sprememba načina delovanja
       "SCADA".alarmi[9] := 1;
       ;
   END_IF;
   #staro_kljuc := "Senzorji_DB".kljuc;



   IF "Senzorji_DB".potiskac_A_koncni_polozaj_zadaj OR "Senzorji_DB".potiskac_A_koncni_polozaj_spredaj THEN
       // Info: Potiskac A na koncnem polozaju
       "SCADA".alarmi[10] := 1;
   ELSE
       "SCADA".alarmi[10] := 0;
   END_IF;

   IF "Senzorji_DB".potiskac_B_koncni_polozaj_zadaj OR "Senzorji_DB".potiskac_B_koncni_polozaj_spredaj THEN
       // Info: Potiskac B na koncnem polozaju
       "SCADA".alarmi[11] := 1;
   ELSE
       "SCADA".alarmi[11] := 0;
   END_IF;

   IF ("Senzorji_DB".potiskac_A_koncni_polozaj_spredaj AND "AutoMotorji".potiskac_A_naprej) OR ("Senzorji_DB".potiskac_A_koncni_polozaj_zadaj AND "AutoMotorji".potiskac_A_nazaj) THEN
       // Error: potiskac A presegel koncen polozaj
       "SCADA".alarmi[12] := 1;
       "Pause_Motors_Flag" := 1;
   END_IF;

   IF ("Senzorji_DB".potiskac_B_koncni_polozaj_spredaj AND "AutoMotorji".potiskac_B_naprej) OR ("Senzorji_DB".potiskac_B_koncni_polozaj_zadaj AND "AutoMotorji".potiskac_B_nazaj) THEN
       // Error: potiskac B presegel koncen polozaj
       "SCADA".alarmi[13] := 1;
       "Pause_Motors_Flag" := 1;
   END_IF;



   IF "SCADA".alarmi[0] AND "SCADA".alarm_potrditev THEN
       "SCADA".alarmi[0] := 0;
       "Pause_Motors_Flag" := 0;
       //muha na lokaciji 2
   END_IF;

   IF "SCADA".alarmi[1] AND "SCADA".alarm_potrditev THEN
       "SCADA".alarmi[1] := 0;
       "Pause_Motors_Flag" := 0;
       //muha na lokaciji 4

   END_IF;

   IF "SCADA".alarmi[2] AND "SCADA".alarm_potrditev THEN
       "SCADA".alarmi[2] := 0;
       "Pause_Motors_Flag" := 0;
       //muha na lokaciji 5

   END_IF;
   IF "SCADA".alarmi[3] AND "SCADA".alarm_potrditev THEN
       "SCADA".alarmi[3] := 0;
       "Pause_Motors_Flag" := 0;
       //muha na lokaciji 7

   END_IF;
   IF "SCADA".alarmi[4] AND "SCADA".alarm_potrditev THEN
       "SCADA".alarmi[4] := 0;
       //prehod l1_l2_predolgo_traja
       //
       "retval":= BLKMOV(SRCBLK:="Lokacije_DB".Empty, DSTBLK=>"Lokacije_DB".L2_vhod_2);
       "retval" := BLKMOV(SRCBLK := "Lokacije_DB".Empty, DSTBLK => "Lokacije_DB".L1_vhod_1);
       "AutoMotorji".trak_A_vhod_naprej := 0;
       "Auto_0_vhod1_DB".Stanje := 0;
       "Pause_Motors_Flag" := 0;



   END_IF;
   IF "SCADA".alarmi[5] AND "SCADA".alarm_potrditev THEN
       "SCADA".alarmi[5] := 0;
       //prehod l2_l4_predolgo_traja
       //
       IF "Auto_1_Potiskac_DB".ID_v_premikanju = "Lokacije_DB".L3_potiskac_A.ID THEN
           "retval" := BLKMOV(SRCBLK := "Lokacije_DB".Empty, DSTBLK => "Lokacije_DB".L3_potiskac_A);
           ;
       END_IF;


       "retval" := BLKMOV(SRCBLK := "Lokacije_DB".Empty, DSTBLK => "Lokacije_DB".L4_naprava_A);
       "AutoMotorji".trak_A_stroj_naprej := 0;
       "AutoMotorji".naprava_A_CCW := 0;
       "AutoMotorji".naprava_A_CW := 0;
       "Auto_1_Potiskac_DB".Stanje := 0;
       "Auto_2_A_Naprava_DB".Stanje := 0;
       "Pause_Motors_Flag" := 0;

   END_IF;
   IF "SCADA".alarmi[6] AND "SCADA".alarm_potrditev THEN
       "SCADA".alarmi[6] := 0;
       //prehod l4_l5_predolgo_traja
       "retval" := BLKMOV(SRCBLK := "Lokacije_DB".Empty, DSTBLK => "Lokacije_DB".L4_naprava_A);
       "retval" := BLKMOV(SRCBLK := "Lokacije_DB".Empty, DSTBLK => "Lokacije_DB".L5_naprava_B);
       "AutoMotorji".trak_A_stroj_naprej := 0;
       "AutoMotorji".trak_B_stroj_naprej := 0;
       "Auto_2_A_Naprava_DB".Stanje := 0;
       "Auto_3_B_Naprava_DB".Stanje := 0;
       "Pause_Motors_Flag" := 0;


   END_IF;

   IF "SCADA".alarmi[7] AND "SCADA".alarm_potrditev THEN
       "SCADA".alarmi[7] := 0;
       //prehod l5_l7_predolgo_traja
       IF "Auto_4_Potiskac_DB".ID_v_premikanju = "Lokacije_DB".L6_potiskac_B.ID THEN
           "retval" := BLKMOV(SRCBLK := "Lokacije_DB".Empty, DSTBLK => "Lokacije_DB".L6_potiskac_B);
       ;
   END_IF;


   "retval" := BLKMOV(SRCBLK := "Lokacije_DB".Empty, DSTBLK => "Lokacije_DB".L7_izhod);
   "AutoMotorji".trak_B_izhod_naprej := 0;

   "Auto_4_Potiskac_DB".Stanje := 0;
   "Auto_5_Izhod_DB".Stanje := 0;
   "Pause_Motors_Flag" := 0;

   END_IF;

   IF "SCADA".alarmi[8] AND "SCADA".alarm_potrditev THEN
       "SCADA".alarmi[8] := 0;
       // Sprememba recepta

   END_IF;

   IF "SCADA".alarmi[9] AND "SCADA".alarm_potrditev THEN
       "SCADA".alarmi[9] := 0;
       // Sprememba načina izvajanja

   END_IF;

   IF "SCADA".alarmi[10] AND "SCADA".alarm_potrditev THEN
       "SCADA".alarmi[10] := 0;
       // Info: Potiskac A na koncnem polozaju

   END_IF;

   IF "SCADA".alarmi[11] AND "SCADA".alarm_potrditev THEN
       "SCADA".alarmi[11] := 0;
       // Info: Potiskac B na koncnem polozaju

   END_IF;

   IF "SCADA".alarmi[12] AND "SCADA".alarm_potrditev THEN
       "SCADA".alarmi[12] := 0;
       "Pause_Motors_Flag" := 0;
       // Error: potiskac A presegel koncen polozaj

   END_IF;
   IF "SCADA".alarmi[13] AND "SCADA".alarm_potrditev THEN
       "SCADA".alarmi[13] := 0;
       "Pause_Motors_Flag" := 0;
       // Error: potiskac B presegel koncen polozaj

   END_IF;
   IF "SCADA".alarmi[14] AND "SCADA".alarm_potrditev THEN
       "SCADA".alarmi[14] := 0;
       "Pause_Motors_Flag" := 0;

       "Startup_Flag" := 0;
       "Ready_Flag" := 1;
       //Naprava ob startu ni v pravilni poziciji

   END_IF;
   IF "SCADA".alarmi[15] AND "SCADA".alarm_potrditev THEN
       "SCADA".alarmi[15] := 0;
       //Naprava polna

   END_IF;
END_FUNCTION_BLOCK

ORGANIZATION_BLOCK "COMPLETE RESTART"   // OB100, SCL
TITLE = "Complete Restart"
{ S7_Optimized_Access := 'FALSE' }
VERSION : 0.1
BEGIN
   IF NOT  "Startup_Flag" THEN
       "Startup_Flag":=1;
   END_IF;
END_ORGANIZATION_BLOCK

// folder: GlavniProgram/SCADA

FUNCTION_BLOCK "SCADAVisual"   // FB11, LAD
{ S7_Optimized_Access := 'FALSE' }
VERSION : 0.1
   VAR_TEMP   // added for the SCL form of the ladder/FBD networks
      _w1 : Bool;
   END_VAR
BEGIN

REGION Network 1
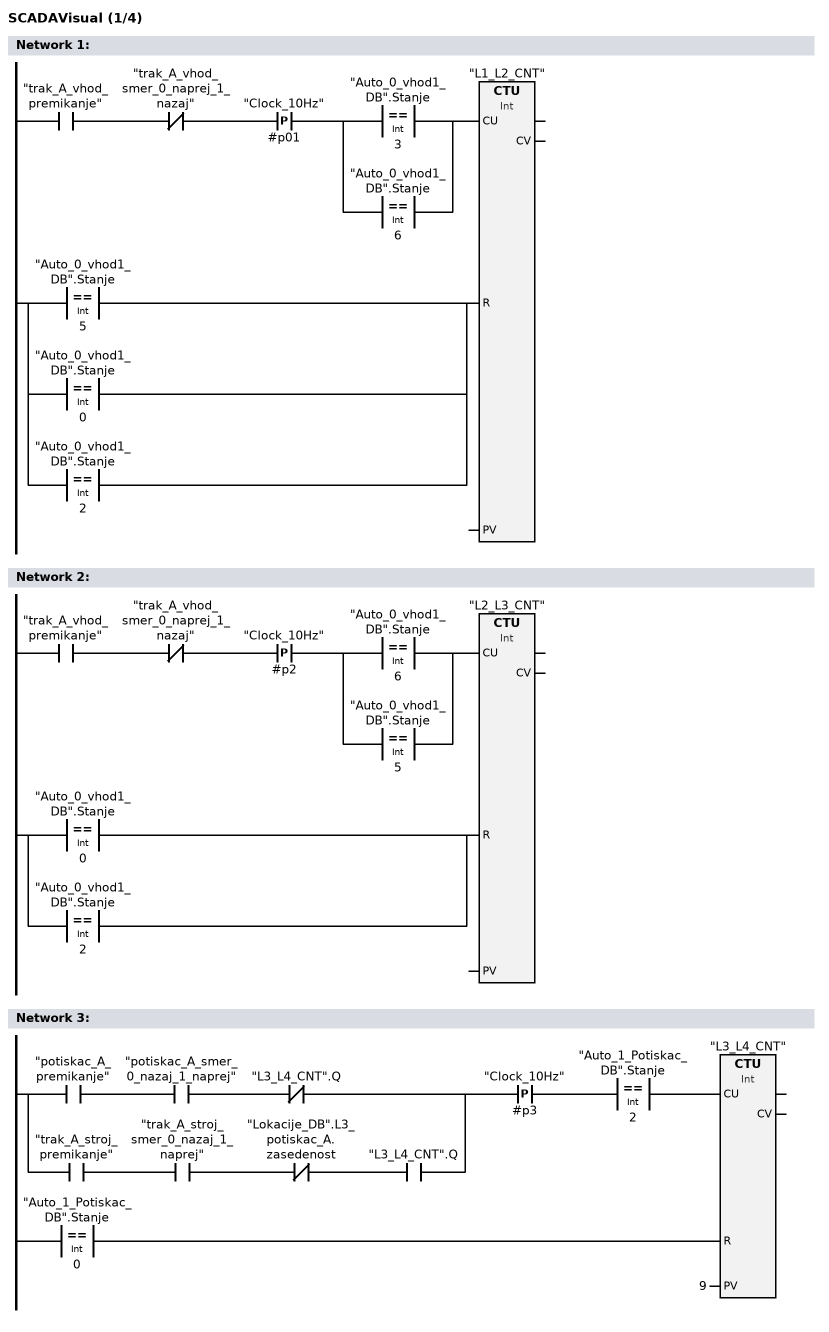
   #_w1 := "trak_A_vhod_premikanje" AND NOT "trak_A_vhod_smer_0_naprej_1_nazaj" AND "Clock_10Hz" AND NOT #p01;   // rising edge of "Clock_10Hz"
   #p01 := "Clock_10Hz";
   "L1_L2_CNT".CTU(CU := #_w1 AND (("Auto_0_vhod1_DB".Stanje = 3) OR ("Auto_0_vhod1_DB".Stanje = 6)),
                   R := ("Auto_0_vhod1_DB".Stanje = 5) OR ("Auto_0_vhod1_DB".Stanje = 0) OR ("Auto_0_vhod1_DB".Stanje = 2));
END_REGION

REGION Network 2
   #_w1 := "trak_A_vhod_premikanje" AND NOT "trak_A_vhod_smer_0_naprej_1_nazaj" AND "Clock_10Hz" AND NOT #p2;   // rising edge of "Clock_10Hz"
   #p2 := "Clock_10Hz";
   "L2_L3_CNT".CTU(CU := #_w1 AND (("Auto_0_vhod1_DB".Stanje = 6) OR ("Auto_0_vhod1_DB".Stanje = 5)),
                   R := ("Auto_0_vhod1_DB".Stanje = 0) OR ("Auto_0_vhod1_DB".Stanje = 2));
END_REGION

REGION Network 3
   #_w1 := (("potiskac_A_premikanje" AND "potiskac_A_smer_0_nazaj_1_naprej" AND NOT "L3_L4_CNT".Q) OR ("trak_A_stroj_premikanje" AND "trak_A_stroj_smer_0_nazaj_1_naprej" AND NOT "Lokacije_DB".L3_potiskac_A.zasedenost AND "L3_L4_CNT".Q)) AND "Clock_10Hz" AND NOT #p3;   // rising edge of "Clock_10Hz"
   #p3 := "Clock_10Hz";
   "L3_L4_CNT".CTU(CU := #_w1 AND ("Auto_1_Potiskac_DB".Stanje = 2),
                   R := "Auto_1_Potiskac_DB".Stanje = 0,
                   PV := 9);
END_REGION

REGION Network 4
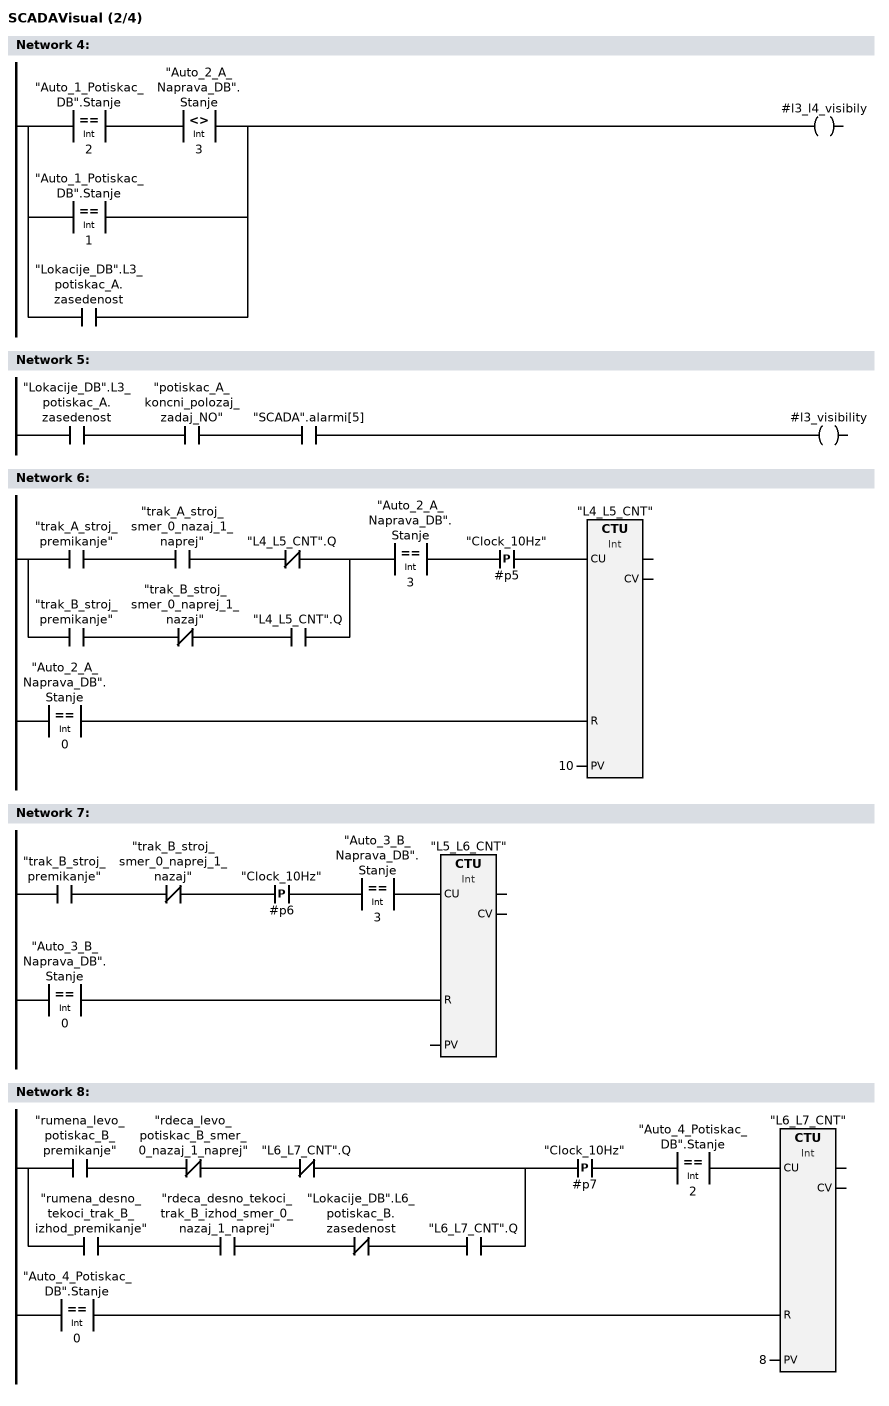
   RUNG wire#powerrail
      { S7_Templates := "SrcType := Int" } EQ_Contact(in1 := "Auto_1_Potiskac_DB".Stanje, in2 := 2)
      { S7_Templates := "SrcType := Int" } NE_Contact(in1 := "Auto_2_A_Naprava_DB".Stanje, in2 := 3)
      wire#w1
      Coil( #l3_l4_visibily )
   END_RUNG
   RUNG wire#powerrail
      { S7_Templates := "SrcType := Int" } EQ_Contact(in1 := "Auto_1_Potiskac_DB".Stanje, in2 := 1)
   END_RUNG wire#w1
   RUNG wire#powerrail
      Contact( "Lokacije_DB".L3_potiskac_A.zasedenost )
   END_RUNG wire#w1
   // the same network as SCL:
   #l3_l4_visibily := (("Auto_1_Potiskac_DB".Stanje = 2) AND ("Auto_2_A_Naprava_DB".Stanje <> 3)) OR ("Auto_1_Potiskac_DB".Stanje = 1) OR "Lokacije_DB".L3_potiskac_A.zasedenost;
END_REGION

REGION Network 5
   RUNG wire#powerrail
      Contact( "Lokacije_DB".L3_potiskac_A.zasedenost )
      Contact( "potiskac_A_koncni_polozaj_zadaj_NO" )
      Contact( "SCADA".alarmi[5] )
      Coil( #l3_visibility )
   END_RUNG
   // the same network as SCL:
   #l3_visibility := "Lokacije_DB".L3_potiskac_A.zasedenost AND "potiskac_A_koncni_polozaj_zadaj_NO" AND "SCADA".alarmi[5];
END_REGION

REGION Network 6
   #_w1 := (("trak_A_stroj_premikanje" AND "trak_A_stroj_smer_0_nazaj_1_naprej" AND NOT "L4_L5_CNT".Q) OR ("trak_B_stroj_premikanje" AND NOT "trak_B_stroj_smer_0_naprej_1_nazaj" AND "L4_L5_CNT".Q)) AND ("Auto_2_A_Naprava_DB".Stanje = 3) AND "Clock_10Hz" AND NOT #p5;   // rising edge of "Clock_10Hz"
   #p5 := "Clock_10Hz";
   "L4_L5_CNT".CTU(CU := #_w1, R := "Auto_2_A_Naprava_DB".Stanje = 0, PV := 10);
END_REGION

REGION Network 7
   #_w1 := "trak_B_stroj_premikanje" AND NOT "trak_B_stroj_smer_0_naprej_1_nazaj" AND "Clock_10Hz" AND NOT #p6;   // rising edge of "Clock_10Hz"
   #p6 := "Clock_10Hz";
   "L5_L6_CNT".CTU(CU := #_w1 AND ("Auto_3_B_Naprava_DB".Stanje = 3), R := "Auto_3_B_Naprava_DB".Stanje = 0);
END_REGION

REGION Network 8
   #_w1 := (("rumena_levo_potiskac_B_premikanje" AND NOT "rdeca_levo_potiskac_B_smer_0_nazaj_1_naprej" AND NOT "L6_L7_CNT".Q) OR ("rumena_desno_tekoci_trak_B_izhod_premikanje" AND "rdeca_desno_tekoci_trak_B_izhod_smer_0_nazaj_1_naprej" AND NOT "Lokacije_DB".L6_potiskac_B.zasedenost AND "L6_L7_CNT".Q)) AND "Clock_10Hz" AND NOT #p7;   // rising edge of "Clock_10Hz"
   #p7 := "Clock_10Hz";
   "L6_L7_CNT".CTU(CU := #_w1 AND ("Auto_4_Potiskac_DB".Stanje = 2),
                   R := "Auto_4_Potiskac_DB".Stanje = 0,
                   PV := 8);
END_REGION

REGION Network 9
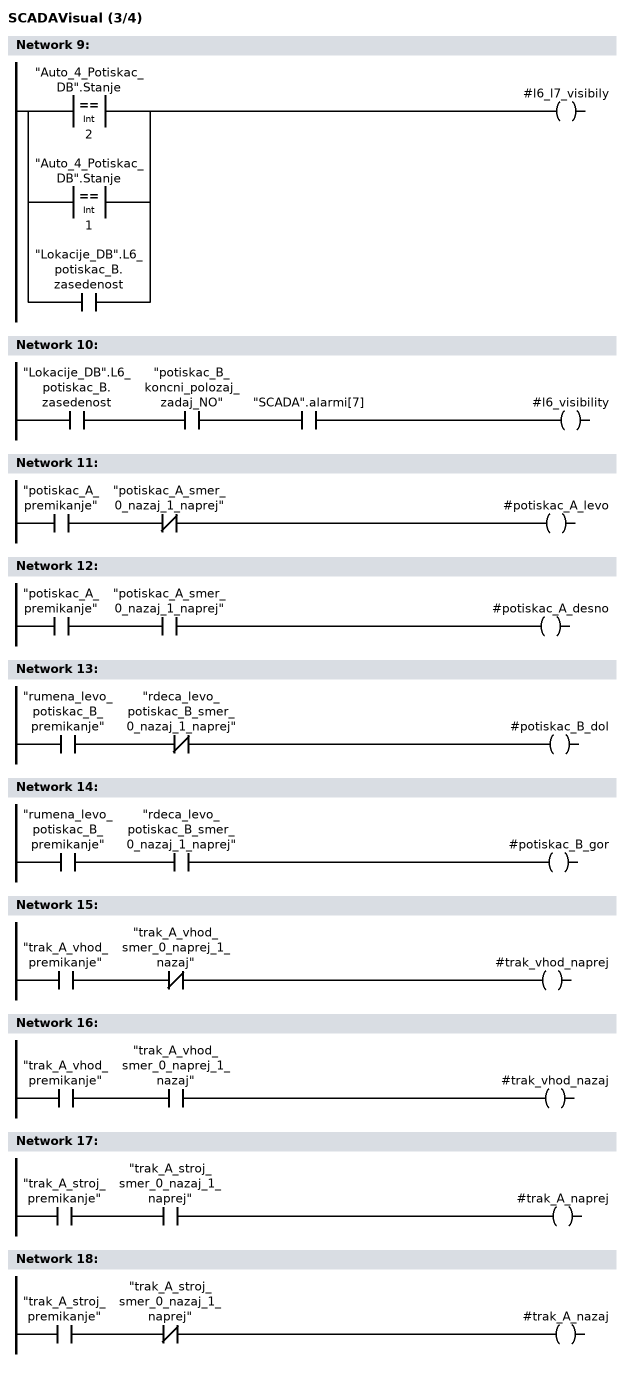
   RUNG wire#powerrail
      { S7_Templates := "SrcType := Int" } EQ_Contact(in1 := "Auto_4_Potiskac_DB".Stanje, in2 := 2)
      wire#w1
      Coil( #l6_l7_visibily )
   END_RUNG
   RUNG wire#powerrail
      { S7_Templates := "SrcType := Int" } EQ_Contact(in1 := "Auto_4_Potiskac_DB".Stanje, in2 := 1)
   END_RUNG wire#w1
   RUNG wire#powerrail
      Contact( "Lokacije_DB".L6_potiskac_B.zasedenost )
   END_RUNG wire#w1
   // the same network as SCL:
   #l6_l7_visibily := ("Auto_4_Potiskac_DB".Stanje = 2) OR ("Auto_4_Potiskac_DB".Stanje = 1) OR "Lokacije_DB".L6_potiskac_B.zasedenost;
END_REGION

REGION Network 10
   RUNG wire#powerrail
      Contact( "Lokacije_DB".L6_potiskac_B.zasedenost )
      Contact( "potiskac_B_koncni_polozaj_zadaj_NO" )
      Contact( "SCADA".alarmi[7] )
      Coil( #l6_visibility )
   END_RUNG
   // the same network as SCL:
   #l6_visibility := "Lokacije_DB".L6_potiskac_B.zasedenost AND "potiskac_B_koncni_polozaj_zadaj_NO" AND "SCADA".alarmi[7];
END_REGION

REGION Network 11
   RUNG wire#powerrail
      Contact( "potiskac_A_premikanje" )
      I_Contact( "potiskac_A_smer_0_nazaj_1_naprej" )
      Coil( #potiskac_A_levo )
   END_RUNG
   // the same network as SCL:
   #potiskac_A_levo := "potiskac_A_premikanje" AND NOT "potiskac_A_smer_0_nazaj_1_naprej";
END_REGION

REGION Network 12
   RUNG wire#powerrail
      Contact( "potiskac_A_premikanje" )
      Contact( "potiskac_A_smer_0_nazaj_1_naprej" )
      Coil( #potiskac_A_desno )
   END_RUNG
   // the same network as SCL:
   #potiskac_A_desno := "potiskac_A_premikanje" AND "potiskac_A_smer_0_nazaj_1_naprej";
END_REGION

REGION Network 13
   RUNG wire#powerrail
      Contact( "rumena_levo_potiskac_B_premikanje" )
      I_Contact( "rdeca_levo_potiskac_B_smer_0_nazaj_1_naprej" )
      Coil( #potiskac_B_dol )
   END_RUNG
   // the same network as SCL:
   #potiskac_B_dol := "rumena_levo_potiskac_B_premikanje" AND NOT "rdeca_levo_potiskac_B_smer_0_nazaj_1_naprej";
END_REGION

REGION Network 14
   RUNG wire#powerrail
      Contact( "rumena_levo_potiskac_B_premikanje" )
      Contact( "rdeca_levo_potiskac_B_smer_0_nazaj_1_naprej" )
      Coil( #potiskac_B_gor )
   END_RUNG
   // the same network as SCL:
   #potiskac_B_gor := "rumena_levo_potiskac_B_premikanje" AND "rdeca_levo_potiskac_B_smer_0_nazaj_1_naprej";
END_REGION

REGION Network 15
   RUNG wire#powerrail
      Contact( "trak_A_vhod_premikanje" )
      I_Contact( "trak_A_vhod_smer_0_naprej_1_nazaj" )
      Coil( #trak_vhod_naprej )
   END_RUNG
   // the same network as SCL:
   #trak_vhod_naprej := "trak_A_vhod_premikanje" AND NOT "trak_A_vhod_smer_0_naprej_1_nazaj";
END_REGION

REGION Network 16
   RUNG wire#powerrail
      Contact( "trak_A_vhod_premikanje" )
      Contact( "trak_A_vhod_smer_0_naprej_1_nazaj" )
      Coil( #trak_vhod_nazaj )
   END_RUNG
   // the same network as SCL:
   #trak_vhod_nazaj := "trak_A_vhod_premikanje" AND "trak_A_vhod_smer_0_naprej_1_nazaj";
END_REGION

REGION Network 17
   RUNG wire#powerrail
      Contact( "trak_A_stroj_premikanje" )
      Contact( "trak_A_stroj_smer_0_nazaj_1_naprej" )
      Coil( #trak_A_naprej )
   END_RUNG
   // the same network as SCL:
   #trak_A_naprej := "trak_A_stroj_premikanje" AND "trak_A_stroj_smer_0_nazaj_1_naprej";
END_REGION

REGION Network 18
   RUNG wire#powerrail
      Contact( "trak_A_stroj_premikanje" )
      I_Contact( "trak_A_stroj_smer_0_nazaj_1_naprej" )
      Coil( #trak_A_nazaj )
   END_RUNG
   // the same network as SCL:
   #trak_A_nazaj := "trak_A_stroj_premikanje" AND NOT "trak_A_stroj_smer_0_nazaj_1_naprej";
END_REGION

REGION Network 19
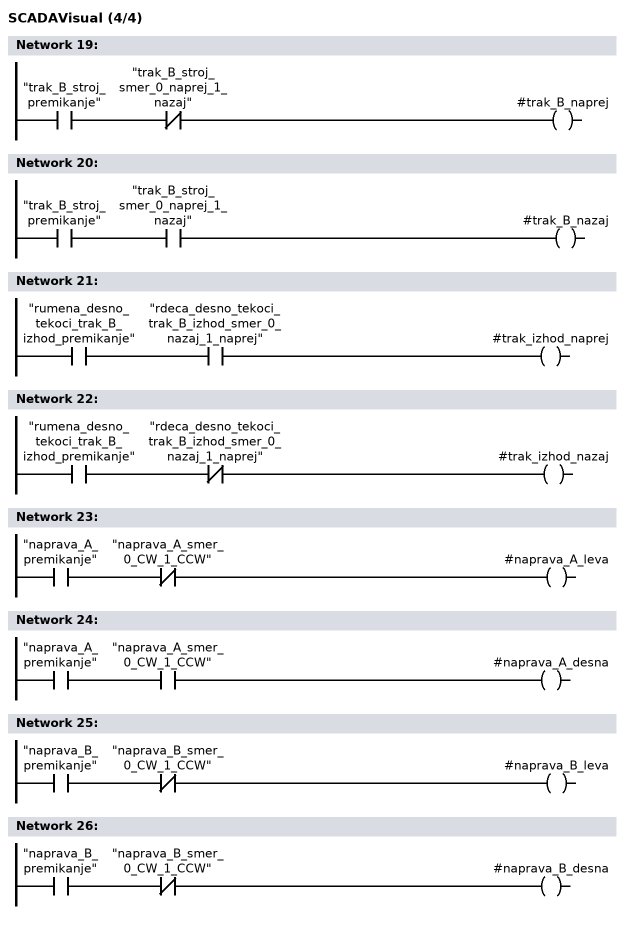
   RUNG wire#powerrail
      Contact( "trak_B_stroj_premikanje" )
      I_Contact( "trak_B_stroj_smer_0_naprej_1_nazaj" )
      Coil( #trak_B_naprej )
   END_RUNG
   // the same network as SCL:
   #trak_B_naprej := "trak_B_stroj_premikanje" AND NOT "trak_B_stroj_smer_0_naprej_1_nazaj";
END_REGION

REGION Network 20
   RUNG wire#powerrail
      Contact( "trak_B_stroj_premikanje" )
      Contact( "trak_B_stroj_smer_0_naprej_1_nazaj" )
      Coil( #trak_B_nazaj )
   END_RUNG
   // the same network as SCL:
   #trak_B_nazaj := "trak_B_stroj_premikanje" AND "trak_B_stroj_smer_0_naprej_1_nazaj";
END_REGION

REGION Network 21
   RUNG wire#powerrail
      Contact( "rumena_desno_tekoci_trak_B_izhod_premikanje" )
      Contact( "rdeca_desno_tekoci_trak_B_izhod_smer_0_nazaj_1_naprej" )
      Coil( #trak_izhod_naprej )
   END_RUNG
   // the same network as SCL:
   #trak_izhod_naprej := "rumena_desno_tekoci_trak_B_izhod_premikanje" AND "rdeca_desno_tekoci_trak_B_izhod_smer_0_nazaj_1_naprej";
END_REGION

REGION Network 22
   RUNG wire#powerrail
      Contact( "rumena_desno_tekoci_trak_B_izhod_premikanje" )
      I_Contact( "rdeca_desno_tekoci_trak_B_izhod_smer_0_nazaj_1_naprej" )
      Coil( #trak_izhod_nazaj )
   END_RUNG
   // the same network as SCL:
   #trak_izhod_nazaj := "rumena_desno_tekoci_trak_B_izhod_premikanje" AND NOT "rdeca_desno_tekoci_trak_B_izhod_smer_0_nazaj_1_naprej";
END_REGION

REGION Network 23
   RUNG wire#powerrail
      Contact( "naprava_A_premikanje" )
      I_Contact( "naprava_A_smer_0_CW_1_CCW" )
      Coil( #naprava_A_leva )
   END_RUNG
   // the same network as SCL:
   #naprava_A_leva := "naprava_A_premikanje" AND NOT "naprava_A_smer_0_CW_1_CCW";
END_REGION

REGION Network 24
   RUNG wire#powerrail
      Contact( "naprava_A_premikanje" )
      Contact( "naprava_A_smer_0_CW_1_CCW" )
      Coil( #naprava_A_desna )
   END_RUNG
   // the same network as SCL:
   #naprava_A_desna := "naprava_A_premikanje" AND "naprava_A_smer_0_CW_1_CCW";
END_REGION

REGION Network 25
   RUNG wire#powerrail
      Contact( "naprava_B_premikanje" )
      I_Contact( "naprava_B_smer_0_CW_1_CCW" )
      Coil( #naprava_B_leva )
   END_RUNG
   // the same network as SCL:
   #naprava_B_leva := "naprava_B_premikanje" AND NOT "naprava_B_smer_0_CW_1_CCW";
END_REGION

REGION Network 26
   RUNG wire#powerrail
      Contact( "naprava_B_premikanje" )
      I_Contact( "naprava_B_smer_0_CW_1_CCW" )
      Coil( #naprava_B_desna )
   END_RUNG
   // the same network as SCL:
   #naprava_B_desna := "naprava_B_premikanje" AND NOT "naprava_B_smer_0_CW_1_CCW";
END_REGION
END_FUNCTION_BLOCK

// folder: MotorLogic

FUNCTION_BLOCK "Izbira_motorja"   // FB1, LAD
TITLE = Izbira motorja s tipkami
{ S7_Optimized_Access := 'FALSE' }
VERSION : 0.1
BEGIN

REGION Network 1: Stevec za izbiro motorja (omejen z 0 in 7)
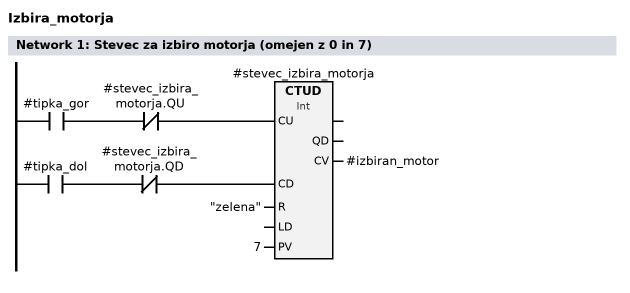
   #stevec_izbira_motorja.CTUD(CU := #tipka_gor AND NOT #stevec_izbira_motorja.QU,
                           CD := #tipka_dol AND NOT #stevec_izbira_motorja.QD,
                           R := "zelena",
                           PV := 7,
                           CV => #izbiran_motor);
END_REGION
END_FUNCTION_BLOCK

FUNCTION_BLOCK "Motor"   // FB2, LAD
TITLE = Vrtenje motorja.
{ S7_Optimized_Access := 'FALSE' }
VERSION : 0.1
BEGIN

REGION Network 1: Časovnik, ki blokira zamenjavo smeri CW za nastavljen čas.
